	13:	IF bAutoModeOn AND  bISealingSeparatorXAxisHome AND  bISealingTopPistonHome AND bISealingBottomPistonHome AND bISealingSeparatorYAxisHome  THEN
		bSaelUnitIntOver:=TRUE;
		step:=step+1;
		END_IF

	14:	bSealingUnitIntOver:=TRUE;
		step:=step+1;



	15:	step:=0;



END_CASE

IF bFwdRevPistonRst THEN bQRForwardPistonValve:=TRUE; bQRReversePistonValve:=TRUE; END_IF

IF bIForwardPistonEnd AND bIReversePistonEnd THEN bFwdRevPistonRst:=FALSE; bQRForwardPistonValve:=FALSE; bQRReversePistonValve:=FALSE; END_IF

IF NOT bIEmergencySwitch OR bStopHmi  OR bServoOff  OR bIMcStop THEN

		bQMWrappingChannelPistonValve1:=FALSE;
		bQMWrappingChannelPistonValve2:=FALSE;
		bQMWrappingChannelPistonValve3:=FALSE;
		bQMForwardPistonValve:=FALSE;
		bQMReversePistonValve:=FALSE;
		bAWrappingCone123OnAuto:=FALSE;
		bAWrappingCone123_23OnAuto:=FALSE;
		bAWrappingCone3OnAuto:=FALSE;
		bAWrappingCone23OnAuto:=FALSE;
		bAWrappingCone23OnAuto1:=FALSE;
		bQAForwardPistonValve:=FALSE;
		bQAReversePistonValve:=FALSE;
		bAInitializeSeq:=FALSE;
		bFwdRevPistonRst:=FALSE;
		bARWrappingCone123OnRst:=FALSE;
		bARWrappingCone123FwdCom:=FALSE;
		bAR3ConeWrappOver:=FALSE;
		tA3ConesealStartDly(IN:=FALSE);
		bQRSealingSeparatorXAxisPistonValve:=FALSE;
		bQRSealingSeparatorYAxisPistonValve:=FALSE;
		bQRSealingTopPistonValve:=FALSE;
		bQRSealingTopPistonValve:=FALSE;
		bSaelUnitIntOver:=FALSE;
		step:=0;

END_IF
END_PROGRAM

(* POU Auto/Sealing_Conveyor_23, ST *)
PROGRAM Sealing_Conveyor_23
VAR

	bA3ConeSealStarted23: BOOL;
	bQASealingConveyor1_23: BOOL;
	bQASealingConveyor2_23: BOOL;
	ConvStopDly1_23: TON;
	bA3ConeSealComp23: BOOL;
	step1: INT;
	CTU_1_23: CTU;
	bAConeCountSenEnable1_23: BOOL;
	bA6thConeSealStarted23: BOOL;
	bA6thConeSealComp23: BOOL;
	ConvStopDly2_23: TON;
	step2: INT;
	step3: INT;
	bSealConvIntOverTemp: BOOL;
	bStopHmitemp: BOOL;
	ConeMissChk_1: RS_Error;
	ConeMissErr_1: BOOL;
	ConeMissChk_2: RS_Error;
	ConeMissErr_2: BOOL;
	ConeMissbit: BOOL;
	SealingStep: INT;
	Timer1: TON;
	Timer2: TON;
	Timer3: TON;
	Timer4: TON;
	bAPauseEnable: BOOL;

	bConeMissBit1: BOOL;
	bConeMissBit2: BOOL;
	bConeMissBit3: BOOL;
	bQASealingConveyor3_23: BOOL;
	tSealStopDly: TIME;
	SealingStep2: INT;
	Timer5: TON;
	Timer6: TON;
	Timer7: TON;
	bConeMissBit11: BOOL;
	bConeMissBit22: BOOL;
	bConeMissBit33: BOOL;
	bConeMissBitSec: BOOL;
	tSealStopDlySec: TIME;
	ConeMissMonitorbit: BOOL;
	bAConeMissAtSealConv: BOOL;
	bAConeMissAtSealConv2: BOOL;
	SingleStep: INT;
	TON_6: TON;
	bAConeCountSenSensed: BOOL;
	bAConeCountSenSensedOff: BOOL;
	R_TRIG_3: R_TRIG;
	R_TRIG_9: R_TRIG;
	CTU_AlarmOnly: CTU;
	bCountLock1: BOOL;
	bCountLock2: BOOL;
	bCountLock: BOOL;
	bAConeMissAtSealConv3: BOOL;
	bQASealingConveyor4_23: BOOL;
	bQASealingConveyor5_23: BOOL;
	bAConeMissAtSealConv4: BOOL;
	bQASealingConveyor6_23: BOOL;
	bCountLock3: BOOL;
	bCountLock4: BOOL;
	bCountLock5: BOOL;
	bCountLock6: BOOL;
	bCountLockBit: BOOL;
	bSet1Started: BOOL;
	bSecSetStarted: BOOL;
	SealCountBit2: BOOL;
END_VAR
bQASealingConveyorMotor2:= ((bQASealingConveyor1_23 OR bQASealingConveyor2_23 OR  bQASealingConveyor3_23 OR bQASealingConveyor5_23 OR bQASealingConveyor4_23 OR bQASealingConveyor6_23 )) ;


CASE step1 OF

	0:	IF bAutoModeOn AND b2_3SetHmiSelected AND   bA3ConeWrappOver AND bQASealingSeparatorYAxisPistonValve THEN
		CTU_1_23.RESET:=TRUE;
		CTU_AlarmOnly.RESET:=TRUE;
		bA3ConeSealStarted23:=TRUE;
		ConvStopDly1_23(IN:=FALSE);
		tSealStopDly:=t#2.5s;
		step1:=step1+1;
		END_IF

	1:	IF NOT bAPauseSeq THEN step1:=step1+1; END_IF


	2:	IF bAutoModeOn AND b2_3SetHmiSelected AND  bA3ConeSealStarted23 AND bISealingSeparatorXAxisEnd THEN
		bA3ConeSealComp23:=TRUE;
		CTU_1_23.RESET:=FALSE;
		CTU_AlarmOnly.RESET:=FALSE;
		 Timer1(IN:=FALSE);
		step1:=step1+1;
		END_IF

	3:	step1:=step1+1;

	4:	IF bAutoModeOn AND   bA3ConeSealComp23  AND (bSealConvStart1 OR bSealConvStart3 ) AND  NOT bAPauseSeq  AND NOT bASealSepaX_axisRsError THEN
		bQASealingConveyor1_23:=TRUE;
		bSet1Started:=TRUE;
		step1:=step1+1;
		END_IF

	5:	ConvStopDly1_23(IN:=FALSE); step1:=step1+1;


	6:	IF CTU_1_23.CV>=3 THEN
		bSealConvStart1:=FALSE;
		bSealConvStart3:=FALSE;
		bA3ConeSealComp23:=FALSE;
		bA3ConeSealStarted23:=FALSE;
		bA3COneCrossed:=TRUE;
		step1:=step1+1;
		END_IF

	7:	step1:=step1+1;

	8:	IF bIColumnconeDetection THEN
		step1:=step1+1;
		END_IF

	9:	step1:=step1+1;


	10:	ConvStopDly1_23(IN:=TRUE , PT:= tSealStopDly , Q=> , ET=> );
		IF ConvStopDly1_23.Q THEN    step1:=step1+1; END_IF


	11:	 step1:=step1+1;

	12:	bQASealingConveyor1_23:=FALSE;
		bA3COneCrossed:=FALSE;
		bQASealingConveyor3_23:=FALSE;
		bQASealingConveyor5_23:=FALSE;
		bQASealingConveyor6_23:=FALSE;
		bAColumnPushPistonStart1_23:=TRUE;
		bASealConvEnd1:=TRUE;
		bCountLock1:=FALSE;
		bCountLock5:=FALSE;
		bCountLock6:=FALSE;
		bSet1Started:=FALSE;
		bCountLockBit:=FALSE;
		step1:=step1+1;

	13:	 step1:=step1+1;


	14:	step1:=0;

END_CASE

IF bQASealingConveyorMotor AND bSet1Started  AND CTU_1_23.CV=3 THEN bCountLockBit:=TRUE; END_IF


IF bQASealingConveyorMotor AND bIConeCountSensor AND b2_3SetHmiSelected AND NOT bCountLockBit AND NOT SealCountBit2  THEN
bAConeCountSenEnable1_23:=TRUE;
ELSE
bAConeCountSenEnable1_23:=FALSE;
END_IF

CTU_1_23(
	CU:=bAConeCountSenEnable1_23 ,
	RESET:= ,
	PV:=6 ,
	Q=> ,
	CV=> );

CTU_AlarmOnly(
	CU:=(bAConeCountSenEnable1_23 AND NOT bCountLock) ,
	RESET:= ,
	PV:=6 ,
	Q=> ,
	CV=> );




CASE step2 OF

	0:	IF bAutoModeOn AND b2_3SetHmiSelected AND  bA6ConeWrappOver23 AND bQASealingSeparatorYAxisPistonValve  THEN
		bA6thConeSealStarted23:=TRUE;
		ConvStopDly2_23(IN:=FALSE);
		tSealStopDlySec:=t#2.5s;
		step2:=step2+1;
		END_IF

	1:	step2:=step2+1;


	2:	 IF   bISealingSeparatorXAxisEnd THEN
		step2:=step2+1;
		END_IF

	3:	 step2:=step2+1;


	4:	IF bAutoModeOn AND b2_3SetHmiSelected  AND bAFirstSetToMatrix   THEN
		bA6thConeSealComp23:=TRUE;
		Timer2(IN:=FALSE); 															(*===============	bAFirstSetToMatrix:=FALSE; ============= Removed for interlock  Checking========= *)
		step2:=step2+1;
		END_IF


	5:	step2:=step2+1;

	6:	IF bAutoModeOn AND   bA6thConeSealComp23  AND  bSealConvStart2 AND  NOT bAPauseSeq THEN
		bQASealingConveyor2_23:=TRUE;
		bSecSetStarted:=TRUE;
		step2:=step2+1;
		END_IF

	7:	ConvStopDly2_23(IN:=FALSE); step2:=step2+1;

	8:	IF CTU_1_23.CV>=6 THEN
		bSealConvStart2:=FALSE;
		bA6thConeSealComp23:=FALSE;
		bA6thConeSealStarted23:=FALSE;
		bA6ConeCrossed:=TRUE;
		step2:=step2+1;
		END_IF

	9:	 step2:=step2+1;

	10:	IF bIColumnconeDetection THEN
		step2:=step2+1;
		END_IF

	11:	 step2:=step2+1;

	12:	ConvStopDly2_23(IN:=TRUE , PT:=tSealStopDlySec , Q=> , ET=> );
		IF ConvStopDly2_23.Q THEN   step2:=step2+1; END_IF

	13:	 step2:=step2+1;

	14:	 CTU_1_23.RESET:=TRUE;
		   step2:=step2+1;

	15:	 step2:=step2+1;

	16:	bQASealingConveyor2_23:=FALSE;
		bQASealingConveyor3_23:=FALSE;
		bQASealingConveyor4_23:=FALSE;
		bA6ConeCrossed:=FALSE;
		bAColumnPushPistonStart2_23:=TRUE;
		bASealConvEnd2:=TRUE;
		bCountLock2:=FALSE;
		bCountLock3:=FALSE;
		bCountLock4:=FALSE;
		SealCountBit2:=FALSE;
		bSecSetStarted:=FALSE;
		  step2:=step2+1;

	17:	 step2:=step2+1;

	18:	CTU_1_23.RESET:=FALSE;
		step2:=0;


END_CASE


IF bQASealingConveyorMotor AND bSecSetStarted AND  CTU_1_23.CV=6 THEN SealCountBit2:=TRUE; END_IF


(*================ Sealing Conveyor Start Condition=============*)


IF bRowStopperIntOver THEN
bSealConvIntOverTemp:=TRUE;
END_IF




CASE step3 OF


0:	IF bSealConvIntOverTemp  AND b2_3SetHmiSelected  THEN
	Step3:=Step3+1;
	END_IF

1:	IF NOT bIColumnconeDetection THEN
	bSealConvStart1:=TRUE;
	Step3:=Step3+1;
	END_IF

2:	IF  CTU_1_23.CV=3 THEN

	Step3:=Step3+1;
	END_IF

3:	IF bIColumnconeDetection THEN
	Step3:=Step3+1;
	END_IF

4:	IF bAFirstSetToMatrix  THEN
	bSealConvStart2:=TRUE;
	Step3:=Step3+1;
	END_IF

5:	IF	CTU_1_23.CV=6 THEN
	bAFirstSetToMatrix:=FALSE;
	Step3:=Step3+1;
	END_IF

6:	IF bIColumnconeDetection THEN
	Step3:=Step3+1;
	END_IF

7:	IF bASecondSetToMatrix THEN
	bSealConvStart3:=TRUE;
	Step3:=Step3+1;
	END_IF

8:	bASecondSetToMatrix:=FALSE;
	Step3:=1;
END_CASE

(*

	IF bSealConvStart1 OR bSealConvStart2 OR bSealConvStart2 THEN
	bAConvReady:=TRUE;
	ELSE
	bAConvReady:=FALSE;
	END_IF
*)
(*=================================Stop Logic=====================*)



IF bQASealingConveyor1_23 AND CTU_AlarmOnly.CV =3  THEN  bCountLock1:=TRUE; END_IF

IF bQASealingConveyor5_23 AND CTU_AlarmOnly.CV =3  THEN  bCountLock5:=TRUE; END_IF

IF bQASealingConveyor6_23 AND CTU_AlarmOnly.CV =3  THEN  bCountLock6:=TRUE; END_IF


IF bQASealingConveyor2_23 AND CTU_AlarmOnly.CV =6  THEN  bCountLock2:=TRUE; END_IF


IF bQASealingConveyor3_23 AND CTU_AlarmOnly.CV =6  THEN  bCountLock3:=TRUE; END_IF


IF bQASealingConveyor4_23 AND CTU_AlarmOnly.CV =6  THEN  bCountLock4:=TRUE; END_IF


 IF bCountLock1 OR bCountLock2 OR  bCountLock3 OR bCountLock4 OR  bCountLock5 OR bCountLock6 THEN bCountLock:=TRUE; ELSE bCountLock:=FALSE; END_IF



IF bQASealingConveyor1_23  AND  bIColumnconeDetection  AND  (CTU_AlarmOnly.CV ) <3  THEN
bAConeMissAtSealConv:=TRUE; SealConeMiss:=' Cone  Missing From Sealing Conveyor';  bQASealingConveyor1_23:=FALSE;  END_IF
(*IF  THEN bAConeMissAtSealConv:=TRUE;  SealConeMiss:=' Cone  Missing From Sealing Conveyor'; bQASealingConveyor1_23:=FALSE; tSealStopDly:=t#4s;
ELSE   SealConeMiss:='Continue Machine Operation'; END_IF *)
IF bAConeMissAtSealConv AND bErrorReset THEN
 bQASealingConveyor5_23:=TRUE;  Step1:=5;  tSealStopDly:=t#4s;    SealConeMiss:='Continue Machine Operation'; bAConeMissAtSealConv:=FALSE; END_IF



IF bQASealingConveyor5_23  AND  bIColumnconeDetection  AND  (CTU_AlarmOnly.CV ) <3  THEN
bAConeMissAtSealConv4:=TRUE; SealConeMiss:=' Cone  Missing From Sealing Conveyor';  bQASealingConveyor5_23:=FALSE;  END_IF
(*IF bQASealingConveyor3_23 AND (CTU_1_23.CV )=3 THEN bAConeMissAtSealConv:=FALSE;  END_IF*)
IF bAConeMissAtSealConv4 AND bErrorReset THEN
bQASealingConveyor6_23:=TRUE;  Step1:=5;  tSealStopDly:=t#4s;    SealConeMiss:='Continue Machine Operation'; bAConeMissAtSealConv4:=FALSE; END_IF




IF bQASealingConveyor2_23 AND  bIColumnconeDetection AND   (CTU_AlarmOnly.CV ) >=3 AND   (CTU_AlarmOnly.CV ) <6 THEN
bAConeMissAtSealConv2:=TRUE; SealConeMiss:=' Cone  Missing From Sealing Conveyor';  bQASealingConveyor2_23:=FALSE;END_IF
(*IF Timer2.Q AND  (CTU_AlarmOnly.CV ) <=6 AND  (CTU_1_23.CV ) >=3 THEN bAConeMissAtSealConv2:=TRUE;  SealConeMiss:=' Cone  Missing From Sealing Conveyor'; bQASealingConveyor2_23:=FALSE; tSealStopDlySec:=t#4s; ELSE   SealConeMiss:='';END_IF*)
IF bAConeMissAtSealConv2 AND bErrorReset THEN
 bQASealingConveyor3_23:=TRUE; Step2:=7; tSealStopDlySec:=t#4s;   SealConeMiss:='Continue Machine Operation'; bAConeMissAtSealConv2:=FALSE; END_IF

(*IF bQASealingConveyor3_23 AND (CTU_1_23.CV )=6 THEN bAConeMissAtSealConv2:=FALSE;  END_IF *)


IF bQASealingConveyor3_23 AND  bIColumnconeDetection AND   (CTU_AlarmOnly.CV ) >=3 AND   (CTU_AlarmOnly.CV ) <6 THEN
  bAConeMissAtSealConv3:=TRUE; SealConeMiss:=' Cone  Missing From Sealing Conveyor';  bQASealingConveyor3_23:=FALSE;END_IF
IF bAConeMissAtSealConv3 AND bErrorReset THEN
 bQASealingConveyor4_23:=TRUE; Step2:=7; tSealStopDlySec:=t#4s;   SealConeMiss:='Continue Machine Operation'; bAConeMissAtSealConv3:=FALSE; END_IF


IF bAConeMissAtSealConv OR bAConeMissAtSealConv3 OR bAConeMissAtSealConv2 OR bAConeMissAtSealConv4  THEN
SealBitAlert:=TRUE; ELSE SealBitAlert:=FALSE; END_IF


IF NOT bIEmergencySwitch OR bStopHmi   OR bServoOff  OR bIMcStop   THEN
CTU_1_23.RESET:=TRUE;
CTU_AlarmOnly.RESET:=TRUE;
ConvStopDly1_23(IN:=FALSE);
bA3ConeSealComp23:=FALSE;
bQASealingConveyor1_23:=FALSE;
bA3COneCrossed:=FALSE;
bAColumnPushPistonStart1_23:=FALSE;
bASealConvEnd1:=FALSE;
bCountLock1:=FALSE;
bCountLock5:=FALSE;
bCountLock6:=FALSE;
bAConeCountSenEnable1_23:=FALSE;
bA6thConeSealStarted23:=FALSE;
ConvStopDly2_23(IN:=FALSE);
bA6thConeSealComp23:=FALSE;
Timer2(IN:=FALSE);
bAColumnPushPistonStart2_23:=FALSE;
bASealConvEnd2:=FALSE;
bCountLock2:=FALSE;
bCountLock3:=FALSE;
bCountLock4:=FALSE;
bSealConvIntOverTemp:=FALSE;
bSealConvStart1:=FALSE;
bSealConvStart2:=FALSE;
bAFirstSetToMatrix:=FALSE;
bSealConvStart3:=FALSE;
bASecondSetToMatrix:=FALSE;
bCountLock:=FALSE;
bAConeMissAtSealConv:=FALSE;
bQASealingConveyor5_23:=FALSE;
bAConeMissAtSealConv4:=FALSE;
bQASealingConveyor6_23:=FALSE;
bQASealingConveyor4_23:=FALSE;
bAConeMissAtSealConv2:=FALSE;
bQASealingConveyor3_23:=FALSE;
SealBitAlert:=FALSE;
bAConeMissAtSealConv3:=FALSE;
step1:=0;
step2:=0;
Step3:=0;

ELSE
CTU_1_23.RESET:=FALSE;
CTU_AlarmOnly.RESET:=FALSE;

END_IF
END_PROGRAM

(* POU Auto1/ConeFeedPiston_23, ST *)
PROGRAM ConeFeedPiston_23
VAR

	R_TRIG_1: R_TRIG;
	CounterTiltRst: BOOL;
	step: INT;

	ConeFeedConvFwdDly1: TON;
	CounterTilt23Rst: BOOL;
	CounterTilt23Rst_R_TRIG: R_TRIG;

	bAConeFeedFwdStart23: BOOL;
	CTU_1: CTU;
	test: BOOL;
	CounterTilt23Enable: BOOL;

	CounterTilt23Rst_TRIG: R_TRIG;

	bIForwardPistonHometemp: BOOL;
	bIReversePistonHometemp: BOOL;
	bITiltingEndtemp: BOOL;
	bITiltingHometemp: BOOL;


	bErrorCheckBit1: BOOL;

	tFwdRSErrCheckDly: TON;
	FwdRevCylHomeChk: RS_Error;
	FwdRevCylHomeSenOk: BOOL;
	FwdRevCylHomeSenErr: BOOL;
	testtemp: BOOL;
	Timer1: TON;
	CTUtEST: CTU;
	CTUtESTcv: INT;
	bAUnitBConeCrossingOff: BOOL;
	step2: INT;
	R_TRIG_3: R_TRIG;
	TON_6: TON;
	bAUnitBConeCrossing_3: BOOL;
	bAUnitBConeCrossingOff_3: BOOL;
	R_TRIG_23: R_TRIG;
	bAfeedingConvOn: BOOL;
END_VAR
IF  NOT bIEmergencySwitch OR bServoOff OR bIMcStop OR   bStopHmi  THEN
	bAConeFeedFwdStart23:=FALSE;
	CounterTiltRst:=TRUE;
	CounterTilt23Rst1:=TRUE;
	bQAConeFeedingPistonOnAuto1:=FALSE;
	CounterTilt23Enable:=FALSE;
	bErrorCheckBit1:=FALSE;
	Timer1(IN:=FALSE);
	FwdRevCylHomeSenOk:=FALSE;
	ConeFeedConvFwdDly1(IN:=FALSE);
	TON_6(IN:= FALSE);
	bAUnitBConeCrossing_3 :=FALSE;
	bAFeedingConvOff:=FALSE;
	step:=0;
	step2:=0;
	ELSE
	CounterTilt23Rst1:=FALSE;
	CounterTiltRst:=FALSE;
END_IF



(*==================== Cone Feeding Piston Logic For 2*3 Model==================*)




IF  b2_3SetHmiSelected AND bAutoModeOn AND ConeFeedConvFwdDly1.Q  AND bIConeFeedingPistonHome   AND  NOT bQAFeedingConveyorMotor
 AND bIForwardPistonHome AND bIReversePistonHome   AND  NOT bAPauseSeq     THEN
		bQAConeFeedingPistonOnAuto1:=TRUE;
END_IF

IF   b2_3SetHmiSelected AND  bQAConeFeedingPistonValve AND bAutoModeOn AND   bIConeFeedingPistonEnd AND  NOT bAPauseSeq
 AND NOT bAConeFeddCylFwdRsError  THEN
		bQAConeFeedingPistonOnAuto1:=FALSE;
END_IF


c18_ConeCounter1(
	CU:=CounterTilt23Enable,
	RESET:=,
	PV:= 18,
	Q=> ,
	CV=> );

CounterTilt23(
	CU:=bAUnitBConeCrossing_3,
	RESET:=CounterTilt23Rst  OR CounterTilt23Rst1,
	PV:= 6,
	Q=> ,
	CV=>CounterTilt23_CV_HMI );
(*

CTUtEST(
	CU:=CounterTilt23Enable ,
	RESET:= ,
	PV:= 56,
	Q=> ,
	CV=>CTUtESTcv );

*)


R_TRIG_23(CLK:=bQAFeedingConveyorMotor , Q=> );
IF R_TRIG_23.Q THEN bAfeedingConvOn:=TRUE; END_IF

IF bIConeOrientationTop  AND b2_3SetHmiSelected AND bQAFeedingConveyorMotor AND bIConeFeedingPistonHome   THEN

CounterTilt23Enable:=TRUE;

ELSE(* IF NOT bAPauseSeq THEN *)
CounterTilt23Enable:=FALSE;
END_IF


R_TRIG_1(CLK:= bIConeOrientationTop , Q=> );


ConeFeedConvFwdDly1(IN:=bAConeFeedFwdStart23 , PT:=t#1s , Q=> , ET=> );  (* ===old Value  PT:=t#1s *)




CASE step OF

	0:	IF CounterTilt23.CV=1AND bIForwardPistonHome AND bIReversePistonHome AND NOT bITiltingEnd  AND bITiltingHome
		AND NOT bAResetEnabled AND bATiltPistonInHome THEN
		bAConeFeedFwdStart23:=TRUE;
		bErrorCheckBit1:=TRUE;
		step:=step+1;
		END_IF sMessage_23_Feeding:='Check Forward , Reverse & Tilting Piston Home Reed Switch ';

	1:	 step:=step+1;

	2:	IF bAutoModeOn AND  bIConeFeedingPistonEnd  AND  NOT bFeedinfCylFwdRsError THEN
		bAConeFeedFwdStart23:=FALSE;
		bATiltPistonInHome:=FALSE;
		bErrorCheckBit1:=FALSE;
		step:=step+1;
		END_IF

	3:	 step:=step+1;

	4:	IF   CounterTilt23.CV = 2  AND bIForwardPistonHome AND bIReversePistonHome  AND bAConeFeedCylStart   AND bITiltingHome AND  NOT bAPauseSeq  THEN
		 bAConeFeedFwdStart23:=TRUE ;
		bErrorCheckBit1:=TRUE;
		IF NOT bIConeFeedingPistonHome THEN
		step:=step+1;
		END_IF
		END_IF sMessage_23_Feeding:='Check Forward , Reverse & Tilting Piston Home Reed Switch ';

	5:	 step:=step+1;

	6:  IF  bAutoModeOn AND bIConeFeedingPistonEnd AND  NOT bFeedinfCylFwdRsError THEN
		bErrorCheckBit1:=FALSE;
		bAConeFeedFwdStart23:=FALSE;
		bAConeFeedCylStart:=FALSE;
		step:=step+1;
		END_IF

	7:	 step:=step+1;


	8:     IF  CounterTilt23.CV = 3 AND bIForwardPistonHome AND bIReversePistonHome AND bITiltingEnd  AND  NOT bAPauseSeq    THEN
		bAConeFeedFwdStart23:=TRUE;
		bErrorCheckBit1:=TRUE;
		step:=step+1;
		END_IF sMessage_23_Feeding:='Check Forward  & Reverse  Piston Home Reed Switch ';

	9:	 step:=step+1;

	10:	IF bAutoModeOn AND  bIConeFeedingPistonEnd AND  NOT bFeedinfCylFwdRsError THEN
		bAConeFeedFwdStart23:=FALSE;
		bErrorCheckBit1:=FALSE;
		step:=step+1;
		END_IF


	11:	step:=step+1;

	12:	IF CounterTilt23.CV = 4 AND bIForwardPistonHome AND bIReversePistonHome    AND bA4thConeFeedStartAuto23
		 AND bITiltingHome  AND  NOT bAPauseSeq   THEN
		bAConeFeedFwdStart23:=TRUE;
		bErrorCheckBit1:=TRUE;
		step:=step+1;
		END_IF sMessage_23_Feeding:='Check Forward ,Reverse & Tilting Piston Home Reed Switch ';

	13:	 step:=step+1;

	14:	IF bAutoModeOn AND  bIConeFeedingPistonEnd AND  NOT bFeedinfCylFwdRsError THEN
		bAConeFeedFwdStart23:=FALSE;
		bErrorCheckBit1:=FALSE;
		bA4thConeFeedStartAuto23:=FALSE;
		step:=step+1;
		END_IF

	15:	step:=step+1;

	16:	IF   CounterTilt23.CV = 5  AND bIForwardPistonHome AND bIReversePistonHome  AND bITiltingEnd    AND  NOT bAPauseSeq    THEN
		bAConeFeedFwdStart23:=TRUE;
		bErrorCheckBit1:=TRUE;
		step:=step+1;
		END_IF sMessage_23:='Check Forward & Reverse Piston Home Reed Switch ';

	17:	 step:=step+1;

	18:	IF bIConeFeedingPistonEnd  AND  NOT bFeedinfCylFwdRsError THEN
		bAConeFeedFwdStart23:=FALSE;
		bErrorCheckBit1:=FALSE;
		step:=step+1;
		END_IF


	19:	Timer1(IN:=FALSE);
		 step:=step+1;



	20: IF   CounterTilt23.CV = 6  AND bIForwardPistonHome AND bIReversePistonHome AND bA6thConeFeedStartAuto23   AND  NOT bAPauseSeq    THEN
		Timer1(IN:=TRUE , PT:=t#0.5s , Q=> , ET=> );
		bErrorCheckBit1:=TRUE;
		IF  Timer1.Q THEN bA6thConeFeedStart23:=FALSE;  step:=step+1; END_IF
		END_IF sMessage_23:='Check Forward  & Reverse   Piston Home Reed Switch ';


	21:	bAConeFeedFwdStart23:=TRUE;
		 step:=step+1;

	22:	IF bIConeFeedingPistonEnd AND  NOT bFeedinfCylFwdRsError THEN
		bAConeFeedFwdStart23:=FALSE;
		Timer1(IN:=FALSE);
		bErrorCheckBit1:=FALSE;
		 step:=step+1;
		END_IF

	23:	step:=step+1;

	24:	CounterTilt23Rst:=TRUE;
		bA6thConeFeedStartAuto23:=FALSE;
		step:=step+1;

	25:	step:=step+1;

	26:	CounterTilt23Rst:=FALSE;
		step:=0;

END_CASE

(*===========Cone crossing sensor single sensing logic for UnitA side======================*)


CASE step2 OF

	0:	R_TRIG_3(CLK:=CounterTilt23Enable , Q=> );
		IF R_TRIG_3.Q THEN TON_6(IN:= FALSE); step2:=step2+1; END_IF


	1:	bAFeedingConvOff:=TRUE; TON_6(IN:= FALSE);
		step2:=step2+1;


	2:	IF NOT bAPauseSeq THEN   bAUnitBConeCrossing_3 :=TRUE;
		 step2:=Step2+1;END_IF

	3:	 step2:=step2+1;

	4: 	TON_6(IN :=  TRUE  , PT:=t#1.3s , Q=> , ET=> );
		IF TON_6.Q THEN  step2:=step2+1; END_IF


	5:	 step2:=step2+1;

	6:	bAUnitBConeCrossingOff_3:=TRUE;
		TON_6(IN:= FALSE);
		step2:=step2+1;

	7:	 step2:=step2+1;

	8:	IF bAUnitBConeCrossingOff_3 THEN bAUnitBConeCrossing_3:=FALSE; step2:=step2+1; END_IF

	9:	IF NOT bAPauseSeq THEN bAUnitBConeCrossingOff_3:=FALSE;
		 step2:=step2+1; END_IF


	10:  IF bIConeFeedingPistonEnd THEN
		step2:=Step2+1; END_IF

	11:	 IF bIConeFeedingPistonHome THEN bAFeedingConvOff:=FALSE; step2:=0; END_IF sMessage_23_Feeding:='Check Cone Feeding Piston Home Reed Switch ';

END_CASE
END_PROGRAM

(* POU Auto1/Tilt_Piston_23, ST *)
PROGRAM Tilt_Piston_23
VAR
	CounterTiltRst: BOOL;
	step: INT;
	bATiltPistonFwdStart23: BOOL;
	test1: BOOL;
	bAConeFeedingStarted23: BOOL;
	bAfeedingCom23: BOOL;
	bAFeedingRev23: BOOL;
	NotbAFeedingRev23: BOOL;
	TiltCylFwdRsErrChk: RS_Error;
	TiltCylFwdRsErr: BOOL;
	bAtiltGoHome2_23temp: BOOL;
END_VAR
	(*===========Cone Tilting Piston Reset Logic===========*)


		IF bRTiltPistonReset  AND bIForwardPistonHome AND bIReversePistonHome THEN
		step:=0;
		CounterTilt23.RESET:=TRUE;
		bATiltPistonFwdStart23:=FALSE;
		bAConeFeedingStarted23:=FALSE;
		bAfeedingCom23:=FALSE;
		bAFeedingRev23:=FALSE;
		NotbAFeedingRev23:=FALSE;
		bA4thConeFeedStartAuto23:=FALSE;
		bA4thConeFeedStart23:=FALSE;;
		bA6thConeFeedStartAuto23:=FALSE;
		bATiltPistonInHome:=FALSE;

		ELSE
		CounterTilt23.RESET:=FALSE;
		END_IF

CASE step OF

	0:	IF  CounterTilt23.CV=1 AND NOT bIConeFeedingPistonEnd AND bIConeFeedingPistonHome   AND bAutoModeOn   AND bIForwardPistonHome AND bIReversePistonHome AND NOT bAPauseSeq   THEN
		bATiltPistonFwdStart23:=FALSE;
		step:=step+1;
		END_IF  sMessage_23_Tilting:='Check Forward and Reverse Piston Home Reed Switch';

	1:	IF bITiltingHome AND NOT bITiltingEnd THEN bATiltPistonInHome:=TRUE; step:=step+1; END_IF

	2: IF  CounterTilt23.CV=2 AND   bAFeedingRev23   AND bIForwardPistonHome AND bIReversePistonHome AND NOT bAPauseSeq
		 AND NOT bAConeFeddCylFwdRsError   THEN
		bATiltPistonFwdStart23:=TRUE;
		step:=step+1;
		END_IF sMessage_23_Tilting:='Check Forward and Reverse Piston Home Reed Switch';

	3:	 step:=step+1;

	4:	 IF  CounterTilt23.CV=3  AND bIForwardPistonHome AND bIReversePistonHome AND NOT bAPauseSeq   THEN
		bATiltPistonFwdStart23:=TRUE;
		step:=step+1;
		END_IF sMessage_23_Tilting:='Check Forward and Reverse Piston Home Reed Switch';

	5:	 step:=step+1;

	6:  IF (* bAtiltGoHome1_23*)  CounterTilt23.CV= 4  AND   bIConeFeedingPistonHome AND bIForwardPistonHome AND bIReversePistonHome
		 AND bATiltEnable1 AND NOT bAPauseSeq    THEN
		bATiltPistonFwdStart23:=FALSE;
		bA4thConeFeedStart23:=TRUE;
		step:=step+1;
		END_IF sMessage_23_Tilting:='Check Forward ,  Reverse & Cone Feeding Piston Home Reed Switch';

	7:	step:=step+1;


	8:  IF  CounterTilt23.CV= 4 AND  bAFeedingRev23 AND bIForwardPistonHome AND bIReversePistonHome AND NOT bAPauseSeq   THEN
		bATiltPistonFwdStart23:=TRUE;
		step:=step+1;
		END_IF  sMessage_23_Tilting:='Check Forward and Reverse Piston Home Reed Switch';

	9:	step:=step+1;


	10:	 bATiltEnable1:=FALSE;
		step:=step+1;


	11:	step:=step+1;

	12:	IF  CounterTilt23.CV=5 AND bIConeFeedingPistonHome AND bIForwardPistonHome AND bIReversePistonHome  AND NOT bAPauseSeq  THEN
		step:=step+1;
		END_IF sMessage_23_Tilting:='Check Forward ,  Reverse & Cone Feeding Piston Home Reed Switch';


	13:	 IF NOT bConeMiss2AtWrapConv THEN  step:=step+1; END_IF

	14:	IF(* bAtiltGoHome2_23 *) CounterTilt23.CV= 6 AND bAtiltGoHome2_23 AND bIForwardPistonHome AND bIReversePistonHome
		 AND bIConeFeedingPistonHome AND NOT bAPauseSeq  AND NOT   bConeMiss2AtWrapConv THEN
		bATiltPistonFwdStart23:=FALSE;
		bA6thConeFeedStart23:=TRUE;
		step:=step+1;
		END_IF  sMessage_23_Tilting:='Check Forward ,  Reverse & Cone Feeding Piston Home Reed Switch';

	15:	 bAtiltGoHome2_23:=FALSE; step:=step+1;



	16:	IF (*CounterTilt23.CV= 6*) b2_3SetHmiSelected  AND bIConeFeedingPistonHome AND bAFeedingRev23  AND bIForwardPistonHome
		 AND bIReversePistonHome AND NOT bAPauseSeq  THEN
		bATiltPistonFwdStart23:=TRUE;
		step:=step+1;
		END_IF  sMessage_23_Tilting:='Check Forward ,  Reverse & Cone Feeding Piston Home Reed Switch';

	17:	 step:=step+1;

	18:	IF bAtiltGoHome3_23 AND bIConeFeedingPistonHome    AND bIForwardPistonHome AND bIReversePistonHome AND NOT bAPauseSeq    THEN
		bATiltPistonFwdStart23:=FALSE;
		step:=0;
		END_IF  sMessage_23_Tilting:='Check Forward ,  Reverse & Cone Feeding Piston Home Reed Switch';


END_CASE


bQAConeTiltingPistonValve2:=bATiltPistonFwdStart23;


IF bQAConeFeedingPistonValve  AND NOT NotbAFeedingRev23 THEN bAConeFeedingStarted23:=TRUE; END_IF

IF bAConeFeedingStarted23 AND bIConeFeedingPistonEnd  AND NOT NotbAFeedingRev23 THEN bAfeedingCom23:=TRUE;  END_IF

IF bAfeedingCom23 AND NOT bIConeFeedingPistonEnd AND NOT NotbAFeedingRev23 THEN bAFeedingRev23:=TRUE;  bAConeFeedingStarted23:=FALSE;   bAfeedingCom23:=FALSE;  END_IF

IF  CounterTilt23.CV= 1 OR  CounterTilt23.CV= 3 OR  CounterTilt23.CV= 5  THEN
NotbAFeedingRev23:=TRUE;
ELSE
NotbAFeedingRev23:=FALSE;
END_IF

IF bATiltPistonFwdStart23  AND bITiltingEnd THEN     bAFeedingRev23:=FALSE; END_IF



IF bA4thConeFeedStart23 AND bITiltingHome THEN
bA4thConeFeedStartAuto23:=TRUE;
END_IF


IF bA6thConeFeedStart23 AND bITiltingHome THEN
bA6thConeFeedStartAuto23:=TRUE;
END_IF
END_PROGRAM

(* POU Auto1/FwdRevPiston_2_3, ST *)
PROGRAM FwdRevPiston_2_3
VAR
	step: INT;
	bA2ndConeReached23: BOOL;
	bA3rdConeReached23: BOOL;
	bA4thConeReached23: BOOL;
	bA5thConeReached23: BOOL;
	bA6thConeReached23: BOOL;
	bA7thConeReached23: BOOL;
	bA8thConeReached23: BOOL;
	bQAForwardPistonValve23: BOOL;
	bQAReversePistonValve23: BOOL;
	test: BOOL;
	FwdCylFwdRSErrChk: RS_Error;
	FwdCylFwdRSErr: BOOL;
	RevCylFwdRSErrChk: RS_Error;
	RevCylFwdRSErr: BOOL;
	FwdCylStartBit1: BOOL;
	FwdCylSTartBit2: BOOL;
	bWrapConvReady: BOOL;
END_VAR
	(*=============================Forward and Reverse piston On/Off logic=======================*)


bQAForwardPistonValve:= ( bQAForwardPistonValve23 );

bQAReversePistonValve:= (bQAReversePistonValve23);


IF bRFwdRevPistonRst OR bAInitializeSeq    THEN
		bQAForwardPistonValve23:=FALSE;
		bQAReversePistonValve23:=FALSE;
		bA2ndConeReached23:=FALSE;
		bInterLocCounterRst:=TRUE;
		bAWrappingConvStart1_23:=FALSE;
		bA2ndConeReached23:=FALSE;
		bA3rdConeReached23:=FALSE;
		bAWrappingConvStart2_23:=FALSE;
		bAtiltGoHome1_23:=FALSE;
		bATiltEnable1:=FALSE;
		bA5thConeReached23:=FALSE;
		bA4thConeReached23:=FALSE;
		bAtiltGoHome2_23:=FALSE;
		bAWrappingConvStart3_23:=FALSE;
		bA6thConeReached23:=FALSE;
		bAtiltGoHome3_23:=FALSE;
		bAWrappingConvStart4_23:=FALSE;
		bA6conesPushedTemp:=FALSE;
		step:=0;


		ELSE
		bInterLocCounterRst:=FALSE;
END_IF




CASE step OF
	0:	IF b2_3SetHmiSelected AND NOT bQAWrappingConveyorMotor  AND NOT bCount_ConvLockBit2 AND bAutoModeOn
		 AND bWrapConvReady  (* AND CounterTilt23.CV=1 AND bITiltingHome AND bIConeFeedingPistonEnd*) AND  NOT bAPauseSeq
		 AND NOT bAConeFeddCylFwdRsError AND NOT bConeMiss4AtWrapConv   THEN
		bQAForwardPistonValve23:=TRUE;
		bInterLocCounterRst:=TRUE;
		bCone1LockBit:=FALSE;
	 (*	bA6conesPushedTemp:=FALSE;  *)
		step:=step+1;
		END_IF


	1:	 step:=step+1;

	2:	IF b2_3SetHmiSelected AND bAutoModeOn AND bIForwardPistonEnd AND  NOT bAPauseSeq AND NOT bAForwPistRsError   THEN
		bQAForwardPistonValve23:=FALSE;
		bWrapConvReady:=FALSE;
		bInterLocCounterRst:=FALSE;
		bAWrappingConvStart1_23:=TRUE;
		step:=step+1;
		END_IF

	3:	 IF  bIForwardPistonHome THEN   bAConeFeedCylStart:=TRUE;  step:=step+1; END_IF
		sMessage_23_Forwad_rev:='Check Forward Piston Home Reed Switch ';


	4:	IF CounterTilt23.CV=2 AND bIConeFeedingPistonEnd  AND  NOT bAPauseSeq  THEN
		bA2ndConeReached23:=TRUE;
	(*	bAWrappingConvStart1_23:=FALSE;  *) (*======== Changed to Wrapping unit_07.10.16=======*)
		step:=step+1;
		END_IF


	5:	 step:=step+1;

	6:	IF CounterTilt23.CV=3 AND bIConeFeedingPistonEnd  AND  NOT bAPauseSeq  THEN
		bA3rdConeReached23:=TRUE;
		step:=step+1;
		END_IF


	7:	 step:=step+1;

	8:	IF b2_3SetHmiSelected AND bAutoModeOn  AND NOT bQAWrappingConveyorMotor  AND bITiltingEnd AND bA2ndConeReached23
		AND bA3rdConeReached23  AND InterLockCounter.CV=1 AND  NOT bAPauseSeq  AND NOT bATiltPistRsError AND NOT bAConeFeddCylFwdRsError
		 AND NOT bAConeMissErrorAtWrpConv AND  NOT bACheckWrappConvError1 THEN
		bQAForwardPistonValve23:=TRUE;
		bQAReversePistonValve23:=TRUE;
		step:=step+1;
		END_IF


	9:	step:= step+1;


	10:	IF b2_3SetHmiSelected AND bAutoModeOn AND bIConeFeedingPistonHome  AND bIForwardPistonEnd AND bIReversePistonEnd
		 AND  NOT bAPauseSeq AND NOT bAForwPistRsError AND NOT bAReversPistnRsError THEN
		bQAForwardPistonValve23:=FALSE;
		bQAReversePistonValve23:=FALSE;
		bA2ndConeReached23:=FALSE;
		bA3rdConeReached23:=FALSE;
		bAWrappingConvStart2_23:=TRUE;
		(*bATiltEnable1:=TRUE;  *)
		step:=step+1;
		END_IF sMessage_23_Forwad_rev:='Check Cone Feeding Piston Home Reed Switch ';

	11:	step:=step+1;

(*-=========================mod Done here & verify============ over==========*)

	12:	 IF b2_3SetHmiSelected AND bAutoModeOn AND bIForwardPistonHome AND bIReversePistonHome  AND  NOT bAPauseSeq   THEN
		bAtiltGoHome1_23:=TRUE;
		bATiltEnable1:=TRUE;
		bAWrappingConvStart2_23:=FALSE;
		step:=step+1;
		END_IF sMessage_23_Forwad_rev:='Check Forward & Reverse Piston Home Reed Switch ';

	13:	step:=step+1;


	14:	IF b2_3SetHmiSelected AND     CounterTilt23.CV=4 AND bIConeFeedingPistonEnd  THEN
		bA4thConeReached23:=TRUE;
		step:=step+1;
		END_IF

	15:	step:=step+1;

	16:	IF b2_3SetHmiSelected AND bAutoModeOn AND NOT bQAWrappingConveyorMotor   AND  bA4thConeReached23
		 AND bITiltingEnd AND bIReversePistonHome THEN
		step:=step+1;
		END_IF sMessage_23_Forwad_rev:='Check Reverse Piston Home Reed Switch ';

	17:	step:=step+1;

	18:	IF  CounterTilt23.CV=5 AND bIConeFeedingPistonEnd THEN
		bA5thConeReached23:=TRUE;
		bAtiltGoHome1_23:=FALSE;
		step:=step+1;
		END_IF

	19:	step:=step+1;

	20:	IF b2_3SetHmiSelected AND bAutoModeOn AND NOT bQAWrappingConveyorMotor  AND( InterLockCounter.CV=3 OR bAByPassOn)
		  AND  bA5thConeReached23 AND bA4thConeReached23  AND bITiltingEnd AND bIReversePistonHome  AND bIForwardPistonHome
		 AND NOT  bATiltPistRsError AND  NOT bAPauseSeq AND NOT bAConeFeddCylFwdRsError  AND NOT bConeMiss2AtWrapConv THEN
		bQAForwardPistonValve23:=TRUE;
		bQAReversePistonValve23:=TRUE;
		step:=step+1;
		END_IF sMessage_23_Forwad_rev:='Check Forward & Reverse Piston Home Reed Switch ';

	21:	step:=step+1;

	22:	IF b2_3SetHmiSelected AND bAutoModeOn AND bIConeFeedingPistonHome  AND bIForwardPistonEnd AND bIReversePistonEnd
		AND  NOT bAPauseSeq AND NOT bAForwPistRsError AND NOT bAReversPistnRsError THEN
		bQAForwardPistonValve23:=FALSE;
		bQAReversePistonValve23:=FALSE;
		bA5thConeReached23:=FALSE;
		bA4thConeReached23:=FALSE;
		bAByPassOn:=FALSE;
		bAWrappingConvStart3_23:=TRUE;
		step:=step+1;
		END_IF sMessage_23_Forwad_rev:='Check Cone Feeding Piston Home Reed Switch ';

	23: step:=step+1;

	24:	IF bAutoModeOn AND bIForwardPistonHome  AND bIReversePistonHome AND  NOT bAPauseSeq THEN
		bAtiltGoHome2_23:=TRUE;
	(*	bAWrappingConvStart3_23:=FALSE;  *)
		step:=step+1;
		END_IF sMessage_23_Forwad_rev:='Check Forward  & Reverse Piston Home Reed Switch ';


	25:	 step:=step+1;


	26:	IF  CounterTilt23.CV=6 AND bIConeFeedingPistonEnd THEN
		bA6thConeReached23:=TRUE;
		step:=step+1;
		END_IF

	27:	step:=step+1;


	28:	IF b2_3SetHmiSelected AND bAutoModeOn AND NOT bQAWrappingConveyorMotor  AND  bA6thConeReached23   AND bITiltingEnd
		  AND bIForwardPistonHome AND( InterLockCounter.CV=5 OR bAByPassOn2 ) AND  NOT bAPauseSeq  AND NOT bATiltPistRsError
		AND NOT bAConeFeddCylFwdRsError AND NOT bConeMiss3AtWrapConv THEN
		bQAReversePistonValve23:=TRUE;
		step:=step+1;
		END_IF sMessage_23_Forwad_rev:='Check Forward Piston Home Reed Switch ';

	29:	 step:=step+1;

	30:	IF b2_3SetHmiSelected AND bAutoModeOn AND bIConeFeedingPistonHome   AND bIReversePistonEnd AND  NOT bAPauseSeq
		 AND NOT  bAReversPistnRsError THEN
		bQAReversePistonValve23:=FALSE;
		bA6thConeReached23:=FALSE;
		bAWrappingConvStart4_23:=TRUE;
		step:=step+1;
		END_IF sMessage_23_Forwad_rev:='Check Cone Feeding Piston Home Reed Switch ';

	31:	step:=step+1;


	32:	IF bAutoModeOn AND bIReversePistonHome THEN
		bAWrappingConvStart4_23:=FALSE;
		bAtiltGoHome3_23:=TRUE;
		step:=step+1;
		END_IF sMessage_23_Forwad_rev:='Check Reverse Piston Home Reed Switch ';

	33:	step:=step+1;

	34:	IF bAutoModeOn AND bITiltingHome THEN
		bAtiltGoHome3_23:=FALSE;
		step:=0;
		END_IF sMessage_23_Forwad_rev:='Check Tilting Piston Home Reed Switch ';
END_CASE

(*======================== InterLock Program for  wrong sensing of sheet or other things when second row Last cone arrived to wrapping conveyor==================*)


IF bCone1LockBit AND bA6conesPushedTemp THEN FwdCylStartBit1:=TRUE; bA6conesPushedTemp:=FALSE;
ELSIF NOT bCone1LockBit AND CounterTilt23.CV=1 AND bITiltingHome AND bIConeFeedingPistonEnd  THEN FwdCylSTartBit2:=TRUE;

END_IF
IF FwdCylStartBit1 OR FwdCylSTartBit2 THEN bWrapConvReady:=TRUE;  FwdCylStartBit1:=FALSE; FwdCylSTartBit2:=FALSE ;   END_IF
END_PROGRAM

(* POU Auto1/ConeFeedConvNew_23, ST *)
PROGRAM ConeFeedConvNew_23
VAR
	bARetUnitRunning: BOOL;
	bConePresentInConv: BOOL;
	tConeFeedConvStopDly: TON;
	step: INT;
	TON_1: TON;
	TON_2: TON;
	TON_3: TON;
	CTU_2: CTU;
	R_TRIG_2: R_TRIG;
	CTU_2Enable: BOOL;
	TON_4: TON;


	R_TRIG_1: R_TRIG;
	TON_5: TON;
	AllOutputsOn: BOOL;
	bAConveStartsAuto: BOOL;
	R_TRIG_3: R_TRIG;
	TON_6: TON;
	bAUnitBConeCrossingOff: BOOL;
	step2: INT;
	testCounter: CTU;
	testreset: BOOL;
	bConeFeedConvRst: BOOL;
	bStopHmitemp: BOOL;
	step3: INT;
	TON_7: TON;
	R_TRIG_4: R_TRIG;
	bAUnitBConeCrossingOff_2: BOOL;
	testCounter_2: CTU;
	i3ConeCountVal: INT;
	CTU_2_UB: CTU;
	i18ConeCountVal: INT;
	bConveyorStarted: BOOL;
	bConePresentInConv_1: BOOL;
END_VAR
bQAFeedingConveyorMotorA:=(bAConveStartsAuto);



IF bMCStartInAuto AND NOT  bIMcStop  AND  bIEmergencySwitch THEN
AllOutputsOn:=TRUE;
ELSE
AllOutputsOn:=FALSE;
END_IF

IF AllOutputsOn(* AND NOT bIConeOrientationTop *) AND NOT bAFeedingConvOff AND NOT bAFeedingConvOff_1  AND bIConeFeedingPistonHome AND NOT bAPauseSeq  THEN
bAConveStartsAuto:=TRUE;
ELSE
bAConveStartsAuto:=FALSE;

END_IF

(*===========Cone crossing sensor single sensing logic for UnitA side======================*)


CASE step2 OF

	0:	R_TRIG_3(CLK:=bIUnitAConeCrossing , Q=> );
		IF R_TRIG_3.Q    THEN TON_6(IN:= FALSE); step2:=step2+1; END_IF


	1:	IF  NOT bAPauseSeq THEN TON_6(IN:= FALSE);
		step2:=step2+1; END_IF


	2:	 bAUnitBConeCrossing_1 :=TRUE;
		 step2:=6;

	3:	 step2:=step2+1;

	4: 	TON_6(IN:=  TRUE  , PT:=t#1ms , Q=> , ET=> );
		IF TON_6.Q    THEN  step2:=step2+1; END_IF


	5:	 step2:=step2+1;

	6:	bAUnitBConeCrossingOff:=TRUE;
		TON_6(IN:= FALSE);
		step2:=step2+1;

	7:	 step2:=step2+1;

	8:	IF bAUnitBConeCrossingOff    THEN bAUnitBConeCrossing_1:=FALSE; step2:=step2+1; END_IF

	9:	 step2:=step2+1;

	10:	bAUnitBConeCrossingOff:=FALSE;
		step2:=0;


END_CASE







testCounter(
	CU:= bAUnitBConeCrossing_1,
	RESET:= ,
	PV:= ,
	Q=> ,
	CV=> );



 (*===============Stop Sequence===========*)


 IF NOT bIEmergencySwitch OR    bStopHmi  OR bIMcStop OR bServoOff  THEN bConeFeedConvRst:=TRUE; ELSE  bConeFeedConvRst:=FALSE;END_IF


IF bConeFeedConvRst THEN
step:=0;
bQAFeedingConveyor1_24:=FALSE;
bQAFeedingConveyor2_24:=FALSE;
bQAFeedingConveyor3_24:=FALSE;
bAConveStartsAuto:=FALSE;
bAUnitBConeCrossingOff:=FALSE;
UnitAConeCrossCount.RESET:=TRUE;
CTU_2.RESET:=TRUE;
step2:=0;
 bAUnitBConeCrossing_1 :=FALSE;
 TON_6(IN:= FALSE);
ELSE
UnitAConeCrossCount.RESET:=FALSE;
CTU_2.RESET:=FALSE;
END_IF



(*==================Logic is to Run the ConeFeed Conveyor Witout Retreival Unit===============*)

IF NOT bAAutoRetrivalEnabled AND bAutoModeOn AND bIMcStart  THEN bStartConeFeedConvInBypass:=TRUE; ELSE bStartConeFeedConvInBypass:=FALSE; END_IF
END_PROGRAM

(* POU Auto/Wrapping_Unit, ST *)
PROGRAM Wrapping_Unit
VAR

	step1: INT;

	R_TRIG_1: R_TRIG;
	Counter1: CTU;
	WrapConvStartDly: TON;
	WrapR_TRIG_1: R_TRIG;
	bAWrappingConvStartAuto2: BOOL;
	WrapR_TRIG_2: R_TRIG;
	WrapConvStartDly2: TON;

	WrapConvStartDly3: TON;
	bAWrappingConvStartAuto3: BOOL;
	WrapR_TRIG_4: R_TRIG;
	bAWrappingConvStartAuto4: BOOL;
	WrapConvStartDly4: TON;
	WrapR_TRIG_5: R_TRIG;
	bAWrappingConvStartAuto5: BOOL;
	WrapConvStartDly5: TON;
	bAWrapConeCyl1: BOOL;
	bAWrapConeCyl3: BOOL;
	bAWrapConeCyl23: BOOL;
	bASet1Comp: BOOL;
	bASet2Comp: BOOL;
	bASet: BOOL;
	bASet3Comp: BOOL;
	bA3ConeWrapStarted: BOOL;
	bA6thConeWrapStarted: BOOL;
	bA1ConeWrappOver: BOOL;
	bA2ConeWrappOver: BOOL;
	bAll3ConeWrapOver: BOOL;
	bA5ConeWrappOver: BOOL;
	bA6ConeWrappOver: BOOL;
	bA56ConeWrapOver: BOOL;
	bAWrapConeCyl23_1: BOOL;

	bATemp: BOOL;
	baConv2ndStart: BOOL;
	baConv3rdStart: BOOL;
	baConv4thStart: BOOL;
	baConv5thStart: BOOL;
	bASensorMonitorBit1: BOOL;
	bAWrappingCone123FwdCom: BOOL;
	ni: BOOL;
	step2: INT;
	bAWrappingCone3FwdCom: BOOL;
	step3: INT;
	bAWrappingCone23FwdCom: BOOL;
	step4: INT;
	bAWrappingCone23FwdCom1: BOOL;
	bASet4Comp: BOOL;
	WrapR_TRIG_3_23: R_TRIG;
	bAWrappingConvStartAuto3_23: BOOL;
	WrapConvStartDly3_23: TON;
	bAWrapConeCyl23_1_23: BOOL;
	bAWrappingCone23_23FwdCom1: BOOL;
	WrapR_TRIG_6_23: R_TRIG;
	bAWrappingConvStartAuto4_23: BOOL;
	WrapConvStartDly6_23: TON;
	bIWrappingCone: BOOL;

	bAWrappingCone123_23FwdCom: BOOL;

	step5: INT;
	bAConvRunning1: BOOL;
	bAConvRunning2: BOOL;
	TON_1: TON;
	TON_2: TON;
	bANextLayerStarted: BOOL;
	bAConvStartInterlock: BOOL;
	bAFirstConeAtWrapConv: BOOL;
	baConveyerStarted: BOOL;
	RtrigBit1: BOOL;
	R_TRIG_3: R_TRIG;
	bASensorNok: BOOL;
	WrapConvStartDlyOver: BOOL;
	test: R_TRIG;
	WrappingCone1RT: R_TRIG;
	WrappingConvRT: R_TRIG;
	WCS1Sensed: BOOL;
	TON_3: TON;
	WCS1SenseRst1: BOOL;
	TON_6: TON;
	TON_7: TON;
	TON_8: TON;
	TON_9: TON;
	TON_10: TON;
	TimerStartBit: BOOL;
	bConvRunning: BOOL;
	test1THEN: BOOL;
	test1: BOOL;
	bSaelUnitIntOverTemp: BOOL;
	step6: INT;
	step7: INT;
	bWCSStart3_24: BOOL;
	bStopHmitemp: BOOL;
	bWCSHomeSenOk: BOOL;
	WCSCylsHomeRsErrChk: RS_Error;
	WCSCylsHomeRsErr: BOOL;
	WCSCylsEndRsErrChk: RS_Error;
	bWCSHomeEndOk: BOOL;
	WCSCylsEndRsErr: BOOL;
	WCSSensorErrChk: RS_Error;
	bAWrappingConvStartAuto3_23temp: BOOL;
	bAWrappingConvStartAuto3_23temp2: BOOL;
	R_Bit1: BOOL;
	R_Bit2: BOOL;
	R_Bit3: BOOL;
	test2: BOOL;
	R_TRIG_2: R_TRIG;
	WCPReadyTemp: BOOL;
	bWrongSenChkBit: BOOL;
	WrapConvOffDly1: TON;
END_VAR
(*========================Wrapping Conveyor Logic in auto Mode=================*)

bQAWrappingConveyorMotor:= (bQAWrappingConveyorMotor1 OR bQAWrappingConveyorMotor2 OR bQAWrappingConveyorMotor3 OR bQAWrappingConveyorMotor4 OR bQAWrappingConveyorMotor5 OR bQAWrappingConveyorMotor3_23 OR bQAWrappingConveyorMotor4_23 );


(*===================Wrapping Pinston On/Off Logic In Auto Mode==================*)


bQAWrappingChannelPistonValve1:= (bAWrappingCone123OnAuto OR bAWrappingCone123_23OnAuto);

bQAWrappingChannelPistonValve2:=( bAWrappingCone123OnAuto OR bAWrappingCone23OnAuto OR bAWrappingCone23OnAuto1 OR bAWrappingCone123_23OnAuto );

bQAWrappingChannelPistonValve3:=( bAWrappingCone123OnAuto OR bAWrappingCone23OnAuto OR bAWrappingCone23OnAuto1 OR  bAWrappingCone3OnAuto OR bAWrappingCone123_23OnAuto  );


(*========================Wrapping Conveyor  Logic for First Cone in auto Mode for 2*4 and 2*3 model=================*)

WrapR_TRIG_1(CLK:= RtrigBit1 , Q=> );


IF  bAWrappingConvStart1 OR bAWrappingConvStart1_23 THEN
RtrigBit1:=TRUE;

ELSE
RtrigBit1:=FALSE;
END_IF


IF bAutoModeOn AND  WrapR_TRIG_1.Q (* OR R_TRIG_3.Q *) AND b2_3SetHmiSelected THEN  bAWrappingConvStartAuto:=TRUE; END_IF

WrapConvStartDly(IN:= bAWrappingConvStartAuto, PT:=t#1s , Q=> , ET=> );




IF bAutoModeOn AND  WrapConvStartDly.Q   AND bIWrappingChannelPiston1_Home AND bIWrappingChannelPiston2_Home
AND bIWrappingChannelPiston3_Home  AND WCPReady AND NOT bIWrappingCone1 AND NOT bIWrappingCone2 AND NOT bIWrappingCone3
AND NOT bACheckWrappConvError1 AND NOT bACheckWrappConvError4  AND b2_3SetHmiSelected  THEN
bQAWrappingConveyorMotor1:=TRUE;
bAconvReayTemp2:=FALSE;
bAconvReadyTemp5:=FALSE;
InterLockCounter.RESET:=FALSE;
bAWrappingConvStartAuto:=FALSE;
bAWrappingConvStart1_23:=FALSE;
bAConvStartBit:=TRUE;
ELSIF bAutoModeOn AND  WrapConvStartDly.Q   AND bIWrappingChannelPiston1_Home AND bIWrappingChannelPiston2_Home AND
bIWrappingChannelPiston3_Home  (*AND bWrongSenChkBit *)AND (  bIWrappingCone1 OR  bIWrappingCone2 OR  bIWrappingCone3 )
 AND NOT bACheckWrappConvError4  AND b2_3SetHmiSelected THEN
bACheckWrappConvError1:=TRUE;
ConeMissAlarm:='Check Wrapping Sensor 1_2_3';
END_IF

IF bACheckWrappConvError1 AND(  bErrorReset OR  bStopHmi ) AND b2_3SetHmiSelected AND NOT bIWrappingCone1 AND NOT  bIWrappingCone2 AND NOT  bIWrappingCone3
THEN  bACheckWrappConvError1:=FALSE; ConeMissAlarm:=''; END_IF

R_TRIG_2(CLK:=bWrpConvIntOver , Q=> );
IF R_TRIG_2.Q THEN WCPReadyTemp:=TRUE; END_IF

IF WCPReadyTemp OR bA6conesPushedTemp THEN bWrongSenChkBit:=TRUE; ELSE  bWrongSenChkBit:=FALSE; END_IF

(*
s
(*==============Wrong Cone or Sheet Sensing Error========================*)


IF  NOT  bCount_ConvLockBitTemp AND   bAutoModeOn AND  bAWrappingConvStartAuto  AND bIWrappingChannelPiston1_Home AND bIWrappingChannelPiston2_Home AND bIWrappingChannelPiston3_Home  AND WCPReady AND(  bIWrappingCone1 OR  bIWrappingCone2 OR  bIWrappingCone3 ) THEN
bACheckWrappConvError1:=TRUE;
(*ConeMissAlarm:='Check Wrapping Sensor 1 & 2 & 3'; *)
END_IF


IF bACheckWrappConvError1 AND  bErrorReset THEN  bACheckWrappConvError1:=FALSE; ConeMissAlarm:=''; END_IF

*)

(*WrapConvOffDly1(IN:= bQAWrappingConveyorMotor1, PT:=t#0.3s , Q=> , ET=> );*)

IF   bAutoModeOn AND  bIWrappingCone1 AND bAConvStartBit  AND b2_3SetHmiSelected  THEN
bQAWrappingConveyorMotor1:=FALSE; END_IF


(*===============Wrapping Conveyor 2nd and 3rd Cone  Logic  in auto Mode for 2*4 and 2*3 model==================*)

(*===============Wrapping piston 1 & 2nd and 3rd  Logic for First Cone in auto Mode  for 2*4 and 2*3 model==================*)

WrapR_TRIG_2(CLK:= ( bAWrappingConvStart2 OR bAWrappingConvStart2_23) , Q=> );


IF bAutoModeOn AND  WrapR_TRIG_2.Q THEN  (* bAWrappingConvStartAuto:=FALSE;  *) bAWrappingConvStartAuto2:=TRUE; END_IF

WrapConvStartDly2(IN:= bAWrappingConvStartAuto2, PT:=t#0.5s , Q=> , ET=> );


IF bAutoModeOn AND  WrapConvStartDly2.Q  AND bIWrappingChannelPiston1_Home AND bIWrappingChannelPiston2_Home
AND bIWrappingChannelPiston3_Home AND NOT bIWrappingCone2 AND NOT bIWrappingCone3  AND NOT bACheckWrappConvError2
AND  b2_3SetHmiSelected THEN
bQAWrappingConveyorMotor2:=TRUE;
bAWrappingConvStartAuto2:=FALSE;
bAConvRunning1:=TRUE;
ELSIF bAutoModeOn AND  WrapConvStartDly2.Q  AND bIWrappingChannelPiston1_Home AND bIWrappingChannelPiston2_Home
AND bIWrappingChannelPiston3_Home AND ( bIWrappingCone2 OR  bIWrappingCone3 ) AND b2_3SetHmiSelected  THEN
bACheckWrappConvError2:=TRUE;
ConeMissAlarm:='Check Wrapping Sensor  2_3';
END_IF

IF bACheckWrappConvError2 AND (bErrorReset  OR  bStopHmi) AND b2_3SetHmiSelected  AND NOT  bIWrappingCone2 AND NOT bIWrappingCone2   THEN bACheckWrappConvError2:=FALSE; ConeMissAlarm:='';  END_IF

IF  bAutoModeOn AND bAConvRunning1  (* AND  bIWrappingCone1 AND bIWrappingCone2   *)AND bIWrappingCone3 THEN
bQAWrappingConveyorMotor2:=FALSE;
  (*bAWrappingConvStartAuto2:=FALSE;  *)
bWrapConvStopped2:=TRUE;
 (*  bAWrapConeCyl123:=TRUE;  *)


END_IF

(*

(*===============Wrong Cone Or Sheet sensing error=====================*)
IF bAutoModeOn AND  bAWrappingConvStartAuto2  AND bIWrappingChannelPiston1_Home AND bIWrappingChannelPiston2_Home AND bIWrappingChannelPiston3_Home AND ( bIWrappingCone2 OR  bIWrappingCone3 ) THEN
bACheckWrappConvError2:=TRUE;
(*ConeMissAlarm:='Check Wrapping Sensor  2 & 3';  *)
END_IF

IF bACheckWrappConvError2 AND bErrorReset THEN bACheckWrappConvError2:=FALSE; ConeMissAlarm:='';  END_IF


*)


(*===============Wrapping piston 123 on/off logic  for 2*4 and 2*3 model =======Cones 1 2 3=============*)
CASE step1 OF

	0:	TON_1(IN:= FALSE);
		step1:=step1+1;

	1:	step1:=step1+1;

	2:	IF bAutoModeOn AND  bAWrapConeCyl123 AND b2_3SetHmiSelected  AND  bIWrappingChannelPiston1_Home   AND bIWrappingChannelPiston2_Home
		 AND bIWrappingChannelPiston3_Home AND NOT bAResetEnabled  AND SealingSafety   THEN
		TON_1(IN:= TRUE, PT:=T#1s , Q=> , ET=> );
		IF TON_1.Q THEN  bAConvRunning1:=FALSE; bAConvStartBit:= FALSE; step1:=step1+1; END_IF
		END_IF

	3:	 step1:=step1+1;


	4:	IF NOT bQASealingConveyorMotor AND NOT bAPauseSeq   AND (  bWCSStart1 OR bWCSStart1_24 OR bWCSStart3 OR bWCSStart3_24 ) AND SealingSafety
		AND bIWrappingCone1 AND bIWrappingCone2 AND bIWrappingCone3 THEN
		bAWrappingCone123OnAuto:=TRUE;
		bA6conesPushedTemp:=FALSE;
		WCPReadyTemp:=FALSE;
		step1:=step1+1;
		END_IF


	5:	 bWCSStart1:=FALSE; bWCSStart3:=FALSE;	step1:=step1+1;


	6:	IF bAWrappingCone123OnAuto AND bIWrappingChannelPiston1_End AND bIWrappingChannelPiston2_End AND bIWrappingChannelPiston3_End
		  AND NOT bAWrap_PistRsError AND bAFilmLoadedCom AND SealingSafety THEN
		bAConvRunning1:=FALSE;
		bAWrappingCone123FwdCom:=TRUE;
		TON_1(IN:= FALSE);
		step1:=step1+1;
		ELSIF  bAWrappingCone123OnAuto AND bIWrappingChannelPiston1_End AND bIWrappingChannelPiston2_End AND bIWrappingChannelPiston3_End
		AND NOT bAWrap_PistRsError  AND NOT bAFilmLoadedCom THEN
		bAFlimNotLoaded:=TRUE;
		bAWrappingCone123OnAuto:=FALSE;
		bAWrapConeCyl123:=FALSE;
		bAPolythinSheetError:=TRUE;
		bSheetNotFeeded:='Sheet NOT Feeded';
		step1:=step1+3;
		END_IF

	7:	  step1:=step1+1;


	8:	 IF bAWrappingCone123FwdCom AND NOT bAPauseSeq  THEN
		bAFilmLoadedCom:=FALSE;
		bAWrappingCone123OnAuto:=FALSE;
		step1:=step1+2;
		END_IF

	9:	 IF bFilmErrClear THEN bSheetNotFeeded:='Continue Machine Operation';  bAFlimNotLoaded:=FALSE;bAConvRunning1:=FALSE;  step1:=step1+1;END_IF

	10:	bAWrapConeCyl123:=FALSE;
		bA3ConeWrappOver:=TRUE;
		step1:=step1+1;

	11:	bFilmErrClear:=FALSE;step1:=step1+1;

	12:	 IF  bIWrappingChannelPiston1_Home   AND bIWrappingChannelPiston2_Home AND bIWrappingChannelPiston3_Home   THEN
		bASet1Comp:=TRUE;
		bAWrappingCone123FwdCom:=FALSE;
		bA3Pushed:=TRUE;
		bCount_ConvLockBit:=FALSE;
		step1:=0;
		END_IF
END_CASE













(*===============Wrapping Conveyor and Piston  4th and 5th Cone  Logic  in auto Mode for 2*3 model==================*)

WrapR_TRIG_3_23(CLK:=bAWrappingConvStart3_23 , Q=> );


IF WrapR_TRIG_3_23.Q THEN bAWrappingConvStartAuto3_23:=TRUE; END_IF


WrapConvStartDly3_23(IN:= bAWrappingConvStartAuto3_23, PT:=t#0.5s , Q=> , ET=> );


IF bAutoModeOn AND  WrapConvStartDly3_23.Q AND  bIWrappingChannelPiston1_Home  AND bIWrappingChannelPiston2_Home
AND bIWrappingChannelPiston3_Home AND  bAconvReayTemp AND NOT bACheckWrappConvError2 AND NOT bACheckWrappConvError3
AND NOT   bIWrappingCone1 AND NOT   bIWrappingCone2 AND NOT bIWrappingCone3  AND b2_3SetHmiSelected  THEN
bQAWrappingConveyorMotor3_23:=TRUE;
bAWrappingConvStart3_23:=FALSE;
bAWrappingConvStartAuto3_23:=FALSE;

ELSIF bAutoModeOn AND  WrapConvStartDly3_23.Q AND  bIWrappingChannelPiston1_Home  AND bIWrappingChannelPiston2_Home
AND bIWrappingChannelPiston3_Home AND  bAconvReayTemp AND (  bIWrappingCone1 OR  bIWrappingCone2 OR bIWrappingCone3 )
AND NOT bACheckWrappConvError2 (*AND NOT bACheckWrappConvError3  *) AND b2_3SetHmiSelected THEN
bACheckWrappConvError3:=TRUE;
ConeMissAlarm:='Check Wrapping Sensor 1_2_3';
END_IF

IF  bASet1Comp AND bQAWrappingConveyorMotor3_23 AND  bAutoModeOn(* AND   bIWrappingCone1*) AND bIWrappingCone2 THEN
bQAWrappingConveyorMotor3_23:=FALSE;
  (*bAWrappingConvStartAuto3_23:=FALSE;  *)  (*==========new modify on 06.10.16==============*)
  bA3Pushed:=FALSE;
bAconvReayTemp:=FALSE;
bWrapConvStopped3:=TRUE;

END_IF
(*

IF bAWrappingConvStartAuto3_23 AND NOT bCount_ConvLockBit AND bIWrappingCone1 THEN R_Bit1:=TRUE ; END_IF

IF bAWrappingConvStartAuto3_23  AND NOT bCount_ConvLockBit AND bIWrappingCone2 THEN R_Bit2:=TRUE;  END_IF

IF bAWrappingConvStartAuto3_23 AND NOT bCount_ConvLockBit  AND bIWrappingCone3 THEN R_Bit3:=TRUE; END_IF


(*===============Wrong Cone Or Sheet sensing error=====================*)
IF  R_Bit1 OR R_Bit2 OR R_Bit3  AND NOT bConeMiss2AtWrapConv  (* AND  bIWrappingChannelPiston1_Home AND bIWrappingChannelPiston2_Home AND bIWrappingChannelPiston3_Home AND *) THEN
bACheckWrappConvError3:=TRUE;
END_IF
*)

IF bACheckWrappConvError3 AND( bErrorReset OR bStopHmi ) AND b2_3SetHmiSelected AND NOT bIWrappingCone1 AND NOT bIWrappingCone2   AND NOT bIWrappingCone3 THEN bACheckWrappConvError3:=FALSE;  END_IF


(*===============Wrapping Conveyor and Piston   6th Cone  Logic  in auto Mode for 2*3 model==================*)

WrapR_TRIG_6_23(CLK:=bAWrappingConvStart4_23 , Q=> );


IF WrapR_TRIG_6_23.Q THEN bAWrappingConvStartAuto4_23:=TRUE; END_IF


WrapConvStartDly6_23(IN:= bAWrappingConvStartAuto4_23, PT:=t#0.5s , Q=> , ET=> );


IF bAutoModeOn AND  WrapConvStartDly6_23.Q AND b2_3SetHmiSelected AND   bIWrappingChannelPiston1_Home AND bIWrappingChannelPiston2_Home
AND bIWrappingChannelPiston3_Home  AND NOT bACheckWrappConvError4 AND NOT bIWrappingCone3  THEN
bQAWrappingConveyorMotor4_23:=TRUE;
bAConvRunning2:=TRUE;
bAWrappingConvStartAuto4_23:=FALSE;
ELSIF  bAutoModeOn AND  WrapConvStartDly6_23.Q AND  bIWrappingChannelPiston1_Home AND bIWrappingChannelPiston2_Home
AND bIWrappingChannelPiston3_Home  AND  bIWrappingCone3 AND b2_3SetHmiSelected  THEN
bACheckWrappConvError4:=TRUE;
ConeMissAlarm:='Check Wrapping Sensor 1_2_3';
bCone1LockBit:=TRUE;
END_IF

IF  bASet1Comp AND  bAutoModeOn AND  bQAWrappingConveyorMotor4_23  AND bAConvRunning2(* AND  bIWrappingCone1 AND bIWrappingCone2  *)
AND bIWrappingCone3 AND b2_3SetHmiSelected  THEN
bQAWrappingConveyorMotor4_23:=FALSE;
bWrapConvStopped4:=TRUE;

(*  bAWrapConeCyl123_23:=TRUE;   *)
END_IF


(*

(*===============Wrong Cone Or Sheet sensing error FOR 6TH Cone=======================*)
IF NOT bCount_ConvLockBit2 AND  bAutoModeOn AND  bAWrappingConvStartAuto4_23 AND  bIWrappingChannelPiston1_Home AND bIWrappingChannelPiston2_Home AND bIWrappingChannelPiston3_Home  AND ( bIWrappingCone1 AND bIWrappingCone2  AND bIWrappingCone3 ) THEN
bACheckWrappConvError4:=TRUE;
bCone1LockBit:=TRUE;
(*ConeMissAlarm:='Check Wrapping Sensor 1 & 2 & 3';*)
END_IF
*)
IF bACheckWrappConvError4 AND ( bErrorReset OR  bStopHmi)   AND NOT  bIWrappingCone3   THEN   bACheckWrappConvError4:=FALSE; ConeMissAlarm:='';  END_IF





(*===============Wrapping piston 123 on/off logic for  2*3 model(4 ,5,6th cone) ====================*)
CASE step5 OF

	0:	TON_2(IN:= FALSE);
		step5:=step5+1;

	1:	step5:=step5+1;

	2:	IF bAutoModeOn AND  bAWrapConeCyl123_23 AND b2_3SetHmiSelected   AND  bIWrappingChannelPiston1_Home   AND bIWrappingChannelPiston2_Home
		 AND bIWrappingChannelPiston3_Home AND NOT bAResetEnabled    THEN
		TON_2(IN:= TRUE, PT:=t#1s , Q=> , ET=> );
		IF TON_2.Q THEN  step5:=step5+1; END_IF
		END_IF

	3:	 step5:=step5+1;

	4:	IF NOT bQASealingConveyorMotor AND bWCSStart2  AND NOT bAPauseSeq AND SealingSafety AND b2_3SetHmiSelected  AND bIWrappingCone1
		AND bIWrappingCone2 AND bIWrappingCone3  THEN
		 bAWrappingCone123_23OnAuto:=TRUE;
		bAByPassOn2:=FALSE;
		 step5:=step5+1;
		END_IF

	5:	bWCSStart2:=FALSE;
		step5:=step5+1;

	6:	IF bAWrappingCone123_23OnAuto AND bIWrappingChannelPiston1_End AND bIWrappingChannelPiston2_End AND bIWrappingChannelPiston3_End
		  AND NOT bAWrap_PistRsError  AND bAFilmLoadedCom AND SealingSafety  AND b2_3SetHmiSelected THEN
		bAConvRunning2:=FALSE;
		bAWrappingCone123_23FwdCom:=TRUE;
		TON_2(IN:= FALSE);

		step5:=step5+1;
		ELSIF  bAWrappingCone123_23OnAuto AND bIWrappingChannelPiston1_End AND bIWrappingChannelPiston2_End AND bIWrappingChannelPiston3_End AND NOT bAWrap_PistRsError  AND NOT bAFilmLoadedCom THEN
		bAFlimNotLoaded:=TRUE;
		bAWrapConeCyl123_23:=FALSE;
		bAPolythinSheetError:=TRUE;
		bSheetNotFeeded:='Sheet NOT Feeded';
		step5:=step5+3;
		END_IF

	7:	 step5:=step5+1;

	8: IF bAWrappingCone123_23FwdCom   AND NOT bAPauseSeq  THEN
		bAWrappingCone123_23OnAuto:=FALSE;
		step5:=step5+2;
		END_IF

	9:	bAWrappingCone123_23OnAuto:=FALSE;
		 IF bFilmErrClear THEN bSheetNotFeeded:='Continue Machine Operation'; bAFlimNotLoaded:=FALSE;bAConvRunning2:=FALSE; step5:=step5+1;END_IF

	10:	bAWrapConeCyl123_23:=FALSE;
		bA6ConeWrappOver23:=TRUE;
		bASet1Comp:=FALSE;
		step5:=step5+1;

	11:	bFilmErrClear:=FALSE;step5:=step5+1;

	12:	 IF  bIWrappingChannelPiston1_Home   AND bIWrappingChannelPiston2_Home AND bIWrappingChannelPiston3_Home   THEN
		bAWrappingCone123_23FwdCom:=FALSE;
		bA6conesPushed:=TRUE;
		bA6conesPushedTemp:=TRUE;
		bCount_ConvLockBitTemp:=FALSE;
		step5:=0;
		END_IF
END_CASE


IF bA6conesPushed AND CounterTilt23.CV<=3 THEN
bANextLayerStarted:=TRUE;
END_IF


IF bA3Pushed OR bA6conesPushed AND bAFirstConeAtWrapConv THEN
bAConvStartInterlock:=TRUE;
ELSE
bAConvStartInterlock:=FALSE;
END_IF

(*

IF bAConvFirstStartUnitB THEN
baConveyerStarted:=TRUE;
END_IF
IF baConveyerStarted AND



*)

WrappingCone1RT(CLK:=( bIWrappingCone1 (*AND bQAWrappingConveyorMotor*) ), Q=> );



WrappingConvRT(CLK:= bQWrappingConveyorMotor , Q=> );

IF  WrappingConvRT.Q THEN
bAWrapConvStarted:=TRUE;

END_IF

IF WrappingCone1RT.Q THEN WCS1Sensed:=TRUE; END_IF

IF WCS1Sensed (*  AND bAWrapConvStarted OR bConvRunning  *)THEN
bAInterlockCountStart:=TRUE;
ELSE
bAInterlockCountStart:=FALSE;
 END_IF



IF  bQWrappingConveyorMotor AND NOT bIWrappingCone1 AND bAutoModeOn THEN
WCS1Sensed:=FALSE;
END_IF

(*

TON_6(IN:=WCS1Sensed , PT:=T#0.2s , Q=> , ET=> );

IF TON_6.Q THEN bAWrapConvStarted:=FALSE; END_IF


IF InterLockCounter.CV = 2 AND bAutoModeOn THEN
TimerStartBit:=TRUE;
bAWrapConvStarted:=FALSE;
TON_10(IN:=TimerStartBit , PT:=t#0.2s , Q=> , ET=> );

 END_IF


IF TON_10.Q AND bQWrappingConveyorMotor THEN
bConvRunning:=TRUE;
END_IF

*)

(*=============== Interlock Logic for  2*3 WCS conveyor===================*)


IF bRowStopperIntOver THEN
bSaelUnitIntOverTemp:=TRUE;
END_IF



CASE step6 OF


0:	IF bSaelUnitIntOverTemp  AND b2_3SetHmiSelected THEN                             (*========= need to check for reset Logic=    step6:=0    =======*)
	Step6:=Step6+1;
	END_IF

1:	bWCSStart1:=TRUE;
	bRowStopperIntOver:=FALSE;
	Step6:=Step6+1;

2:	IF  bASealConvEnd1 THEN
	bSaelUnitIntOverTemp:=FALSE;
	Step6:=Step6+1;
	END_IF

3:	bWCSStart2:=TRUE;
	bASealConvEnd1:=FALSE;
	Step6:=Step6+1;


4:	IF bASealConvEnd2  THEN
	Step6:=Step6+1;
	END_IF

5:	bWCSStart3:=TRUE;
	bASealConvEnd2:=FALSE;
	Step6:=2;

END_CASE


(*
(*=============== Interlock Logic for  2*4 WCS conveyor===================*)


CASE step7 OF


0:	IF bSaelUnitIntOverTemp AND b2_4SetHmiSelected  THEN                                    (*========= need to check for reset Logic=    step7:=0    =======*)
	Step7:=Step7+1;
	END_IF

1:	bWCSStart1_24:=TRUE;
	Step7:=Step7+1;

2:	IF  bASealConvEnd1_24 THEN
	bSaelUnitIntOverTemp:=FALSE;
	Step7:=Step7+1;
	END_IF

3:	bWCSStart2_24:=TRUE;
	bASealConvEnd1_24:=FALSE;
	Step7:=Step7+1;


4:	IF bASealConvEnd2_24  THEN
	Step7:=Step7+1;
	END_IF

5:	bWCSStart3_24:=TRUE;
	bASealConvEnd2_24:=FALSE;
	Step7:=2;

END_CASE

*)

IF NOT bIEmergencySwitch OR bStopHmi  OR bServoOff OR bIMcStop THEN
bAWrappingConvStartAuto3_23:=FALSE;
bAWrappingConvStartAuto4_23:=FALSE;
bAWrappingConvStart4_23:=FALSE;
bAWrappingConvStartAuto:=FALSE;
bQAWrappingConveyorMotor1:=FALSE;
bAWrappingConvStartAuto2:=FALSE;
bQAWrappingConveyorMotor2:=FALSE;
bQAWrappingConveyorMotor3:=FALSE;
bQAWrappingConveyorMotor4:=FALSE;
bQAWrappingConveyorMotor5:=FALSE;
WrapConvStartDly3_23(IN:= FALSE);
bAConvRunning1:=FALSE;
bASet1Comp:=FALSE;
bAWrappingConvStartAuto3:=FALSE;
bAWrapConeCyl3:=FALSE;
bAWrapConeCyl123:=FALSE;
WCS1Sensed:=FALSE;
bAWrappingConvStart1_23:=FALSE;
bSaelUnitIntOver:=FALSE;
bWCSStart1:=FALSE;
bWCSStart2:=FALSE;
bWCSStart3:=FALSE;
bASealConvEnd1:=FALSE;
bASealConvEnd2:=FALSE;
InterLockCounter.RESET:=TRUE;
bAWrappingCone123OnAuto:=FALSE;
bAWrappingCone123_23OnAuto:=FALSE;
bQAWrappingConveyorMotor4_23:=FALSE;
bQAWrappingConveyorMotor3_23:=FALSE;
bCount_ConvLockBit2:=FALSE;
bCount_ConvLockBit:=FALSE;
step1:=0;
step2:=0;
step3:=0;
step4:=0;
step5:=0;
step6:=0;
ELSE
InterLockCounter.RESET:=FALSE;
END_IF
END_PROGRAM

(* POU Auto1/Tilt_Piston_24, ST *)
PROGRAM Tilt_Piston_24
VAR
	CounterTiltRst: BOOL;
	step: INT;
	bATiltPistonFwdStart: BOOL;
	test1: BOOL;
	bAConeFeedingStarted: BOOL;
	bAfeedingCom: BOOL;
	bAFeedingRev: BOOL;
	NotbAFeedingRev: BOOL;
	RstStep: INT;
END_VAR
		IF bRTiltPistonReset  AND bIForwardPistonHome AND bIReversePistonHome THEN
		step:=0;
		bATiltPistonFwdStart:=FALSE;
		bAConeFeedingStarted:=FALSE;
		bAfeedingCom:=FALSE;
		bAFeedingRev:=FALSE;
		NotbAFeedingRev:=FALSE;
		bA4thConeFeedStartAuto23:=FALSE;
		bA4thConeFeedStart23:=FALSE;;
		bA6thConeFeedStartAuto23:=FALSE;
		bATiltPistonInHome:=FALSE;
		bA5thConeFeedStart:=FALSE;
		END_IF




bQAConeTiltingPistonValve1:=bATiltPistonFwdStart;


IF bQAConeFeedingPistonValve  AND NOT NotbAFeedingRev THEN bAConeFeedingStarted:=TRUE; END_IF

IF bAConeFeedingStarted AND bIConeFeedingPistonEnd  AND NOT NotbAFeedingRev THEN bAfeedingCom:=TRUE;  END_IF

IF bAfeedingCom AND NOT bIConeFeedingPistonEnd AND NOT NotbAFeedingRev THEN bAFeedingRev:=TRUE;  bAConeFeedingStarted:=FALSE;   bAfeedingCom:=FALSE;  END_IF

IF  CounterTilt.CV= 1 OR  CounterTilt.CV= 3 OR  CounterTilt.CV= 6 OR  CounterTilt.CV= 8 THEN
NotbAFeedingRev:=TRUE;
ELSE
NotbAFeedingRev:=FALSE;
END_IF

IF bATiltPistonFwdStart  AND bITiltingEnd THEN     bAFeedingRev:=FALSE; END_IF



	                                                                        (*===========Cone Tilting Piston Reset Logic===========*)

CASE step OF

	0:	IF  CounterTilt.CV=1 AND NOT bIConeFeedingPistonEnd    AND bAutoModeOn   AND bIForwardPistonHome AND bIReversePistonHome  THEN
		bATiltPistonFwdStart:=FALSE;  step:=step+1;  END_IF
		 sMessage_23_Tilting:='Check Forward and Reverse Piston Home Reed Switch';


	1:	IF NOT bAPauseSeq THEN  step:=step+1;   END_IF                                (* Cone 1 Logic  Over*)



	2:	 IF  CounterTilt.CV=2 AND   bAFeedingRev   AND bIForwardPistonHome AND bIReversePistonHome AND bIConeFeedingPistonHome  THEN
		bATiltPistonFwdStart:=TRUE;
		bATiltEnable1_24:=FALSE; step:=step+1; END_IF
		sMessage_23_Tilting:='Check Forward ,  Reverse & Cone Feeding Piston Home Reed Switch';

	3:	IF NOT bAPauseSeq THEN step:=step+1; END_IF                                   (* Cone 2 Logic  Over*)



	4:	 IF  CounterTilt.CV=3  AND bIForwardPistonHome AND bIReversePistonHome  AND bIConeFeedingPistonHome  THEN
		bATiltPistonFwdStart:=TRUE; step:=step+1;END_IF
		 sMessage_23_Tilting:='Check Forward ,  Reverse & Cone Feeding Piston Home Reed Switch';


	5:	IF NOT bAPauseSeq THEN step:=step+1; END_IF

	6:	  IF (* CounterTilt.CV=4 *) bATiltEnable2_24 AND   bIConeFeedingPistonHome AND bIForwardPistonHome AND bIReversePistonHome THEN
		bATiltPistonFwdStart:=FALSE;step:=step+1; END_IF
		sMessage_23_Tilting:='Check Forward ,  Reverse & Cone Feeding Piston Home Reed Switch';


	7:	IF NOT bAPauseSeq THEN step:=step+1; END_IF                               (* Cone 3 Logic  Over*)




	8:  IF  CounterTilt.CV= 4 AND  bAFeedingRev AND bIForwardPistonHome AND bIReversePistonHome   THEN
		bATiltPistonFwdStart:=TRUE;
		bATiltEnable2_24:=FALSE; step:=step+1; END_IF
		 sMessage_23_Tilting:='Check Forward and Reverse Piston Home Reed Switch';

	9:	IF NOT bAPauseSeq THEN step:=step+1; END_IF

	10:  IF bAtiltGoHome THEN
		bATiltPistonFwdStart:=FALSE;
		bA5thConeFeedStart:=TRUE;
		step:=step+1;
		END_IF

	11:	IF NOT bAPauseSeq THEN step:=step+1; END_IF                           (* Cone 4 Logic  Over*)




	12:	IF  CounterTilt.CV=5 AND bIConeFeedingPistonHome AND bIForwardPistonHome AND bIReversePistonHome   THEN
		bATiltPistonFwdStart:=FALSE; step:=step+1; END_IF
		sMessage_23_Tilting:='Check Forward ,  Reverse & Cone Feeding Piston Home Reed Switch';


	13:	IF NOT bAPauseSeq THEN step:=step+1; END_IF

	14:	IF CounterTilt.CV= 5 AND    bAFeedingRev AND bIForwardPistonHome AND bIReversePistonHome THEN
		bATiltPistonFwdStart:=TRUE; step:=step+1; END_IF
		 sMessage_23_Tilting:='Check Forward and Reverse Piston Home Reed Switch';

	15:	IF NOT bAPauseSeq THEN step:=step+1; END_IF

	16:	step:=step+1;

	17:	IF NOT bAPauseSeq THEN step:=step+1; END_IF                           (* Cone 5 Logic  Over*)





	18:	IF CounterTilt.CV= 6 AND bIConeFeedingPistonHome   AND bIForwardPistonHome AND bIReversePistonHome THEN
		step:=step+1; END_IF
		sMessage_23_Tilting:='Check Forward ,  Reverse & Cone Feeding Piston Home Reed Switch';

	19:	IF NOT bAPauseSeq THEN step:=step+1; END_IF

	20:	IF(* CounterTilt.CV= 7 *) bATiltEnable3_24  AND bIConeFeedingPistonHome    AND bIForwardPistonHome AND bIReversePistonHome THEN
		bATiltPistonFwdStart:=FALSE; step:=step+1; END_IF
		sMessage_23_Tilting:='Check Forward ,  Reverse & Cone Feeding Piston Home Reed Switch';


	21:	IF NOT bAPauseSeq THEN step:=step+1; END_IF                           (* Cone 6 Logic  Over*)





	22:	IF CounterTilt.CV= 7 AND bAFeedingRev    AND bIForwardPistonHome AND bIReversePistonHome THEN
		bATiltPistonFwdStart:=TRUE;
		bATiltEnable3_24:=FALSE; step:=step+1; END_IF
		 sMessage_23_Tilting:='Check Forward and Reverse Piston Home Reed Switch';

	23:	IF NOT bAPauseSeq THEN step:=step+1; END_IF

	24:	IF (* CounterTilt.CV= 1*) bATiltEnable1_24  AND bIConeFeedingPistonHome    AND bIForwardPistonHome AND bIReversePistonHome THEN
		bATiltPistonFwdStart:=FALSE; step:=0; END_IF
		sMessage_23_Tilting:='Check Forward ,  Reverse & Cone Feeding Piston Home Reed Switch';


                                                                                                                                              (* Cone 7 Logic  Over*)

END_CASE






(*
		(*===========Cone Tilting Piston On/Off Logic===========*)


		IF     bAutoModeOn AND  bConeEvenCount AND bIConeFeedingPistonEnd AND bIForwardPistonHome AND bIReversePistonHome AND NOT  bIForwardPistonEnd AND NOT  bIReversePistonEnd THEN
		bQAConeTiltingPistonValve:=TRUE;
		END_IF

		IF   bAutoModeOn AND CounterTilt.CV=4 AND  bIConeFeedingPistonHome AND bIForwardPistonHome AND bIReversePistonHome AND NOT  bIForwardPistonEnd AND NOT  bIReversePistonEnd   THEN
		bQAConeTiltingPistonValve:=FALSE;
		END_IF


*)
END_PROGRAM

(* POU Auto1/FwdRevPiston_2_4, ST *)
PROGRAM FwdRevPiston_2_4
VAR
	step: INT;
	bA2ndConeReached: BOOL;
	bA3rdConeReached: BOOL;
	bA4thConeReached: BOOL;
	bA5thConeReached: BOOL;
	bA6thConeReached: BOOL;
	bA7thConeReached: BOOL;
	bA8thConeReached: BOOL;
	fs: BOOL;
END_VAR
	                             (*=============================Forward and Reverse piston On/Off logic For 2*4 model=======================*)



CASE step OF


	 0:	 IF CounterTilt.CV=1 AND bIConeFeedingPistonEnd  THEN bAFirstConeReached:=TRUE; step:=step+1; END_IF

	 1:	 IF NOT bAPauseSeq THEN step:=step+1; END_IF

 	 2:  	IF b2_4SetHmiSelected AND NOT bQAWrappingConveyorMotor AND NOT bACheckWrappConvError5 AND
		 bAutoModeOn  AND bAFirstConeReached AND bITiltingHome AND  InterLockCounter.CV = 0 AND NOT bAPauseSeq  THEN
		bQAForwardPistonValve:=TRUE; step:=step+1; END_IF

	 3:	IF NOT bAPauseSeq THEN step:=step+1; END_IF

	 4:	IF b2_4SetHmiSelected AND bAutoModeOn AND bIForwardPistonEnd AND NOT bAPauseSeq THEN
		bA8thoneReachecdWCS:=FALSE;
		bQAForwardPistonValve:=FALSE;
		bAFirstConeReached:=FALSE;
		bAWrappingConvStart1:=TRUE;
		bAConeFeedPistonLockOk:=TRUE; step:=step+1;END_IF

	5:     IF NOT bAPauseSeq THEN step:=step+1; END_IF                                                (* Cone 1 Logic  Over*)




	6:	IF CounterTilt.CV=2 AND bIConeFeedingPistonEnd  AND NOT bAPauseSeq  THEN
		bA2ndConeReached:=TRUE;
		(*bAWrappingConvStart1:=FALSE;*) step:=step+1; END_IF

	7:	IF NOT bAPauseSeq THEN step:=step+1; END_IF                                              (* Cone 2 Logic  Over*)




	8:	IF CounterTilt.CV=3 AND bIConeFeedingPistonEnd  AND  NOT bAPauseSeq THEN
		bA3rdConeReached:=TRUE; step:=step+1; END_IF

	9:	IF NOT bAPauseSeq THEN step:=step+1; END_IF

	10:	IF b2_4SetHmiSelected AND bAutoModeOn AND NOT bACheckWrappConvError1 AND NOT bQAWrappingConveyorMotor
		AND bITiltingEnd AND bA2ndConeReached AND bA3rdConeReached AND InterLockCounter.CV=1 AND NOT bAPauseSeq  THEN
		bQAForwardPistonValve:=TRUE;
		bQAReversePistonValve:=TRUE; step:=step+1; END_IF

	11:	IF NOT bAPauseSeq THEN step:=step+1; END_IF

	12:	IF b2_4SetHmiSelected AND bAutoModeOn AND bIConeFeedingPistonHome  AND bIForwardPistonEnd AND bIReversePistonEnd AND   NOT bAPauseSeq   THEN
		bQAForwardPistonValve:=FALSE;
		bQAReversePistonValve:=FALSE;
		bA2ndConeReached:=FALSE;
		bA3rdConeReached:=FALSE;
		bAWrappingConvStart2:=TRUE;
		bATiltEnable2_24 := TRUE; step:=step+1; END_IF

	13:	IF NOT bAPauseSeq THEN step:=step+1; END_IF                                                  (* Cone 3 Logic  Over*)




                                                                     (*-=========================mod need here=======================*)
	14:	IF  CounterTilt.CV=4 AND bIConeFeedingPistonEnd THEN
		bA4thConeReached:=TRUE;
		(*bAWrappingConvStart2:=FALSE;*) step:=step+1; END_IF

	15:	IF NOT bAPauseSeq THEN step:=step+1; END_IF

	16:	IF b2_4SetHmiSelected AND bAutoModeOn AND NOT bACheckWrappConvError2 AND NOT bQAWrappingConveyorMotor
		AND  bA4thConeReached  AND bITiltingEnd AND bIReversePistonHome AND  InterLockCounter.CV=3  AND NOT bAPauseSeq  THEN
		bQAReversePistonValve:=TRUE; step:=step+1; END_IF

	17:	IF NOT bAPauseSeq THEN step:=step+1; END_IF

	18:	IF b2_4SetHmiSelected AND bAutoModeOn AND bIReversePistonEnd  AND bITiltingEnd   AND NOT bAPauseSeq THEN
		bQAReversePistonValve:=FALSE;
		bA4thConeReached:=FALSE;
		bAWrappingConvStart3:=TRUE; step:=step+1; END_IF

	19:	IF NOT bAPauseSeq THEN step:=step+1; END_IF

	20:	 IF b2_4SetHmiSelected AND bAutoModeOn AND bIReversePistonHome  AND NOT bAPauseSeq  THEN
		bAtiltGoHome:=TRUE;
		(*bAWrappingConvStart3:=FALSE;*) step:=step+1; END_IF

	21:	IF NOT bAPauseSeq THEN step:=step+1; END_IF                                                             (* Cone 4 Logic  Over*)




	22:	IF  CounterTilt.CV=5 AND bIConeFeedingPistonEnd THEN
		bA5thConeReached:=TRUE;
		bAtiltGoHome:=FALSE; step:=step+1; END_IF

	23:	IF NOT bAPauseSeq THEN step:=step+1; END_IF                                                               (* Cone 5 Logic  Over*)




	24:	IF CounterTilt.CV=6 AND bIConeFeedingPistonEnd  THEN
		bA6thConeReached:=TRUE; step:=step+1; END_IF

	25:	IF NOT bAPauseSeq THEN step:=step+1; END_IF

	26:	IF b2_4SetHmiSelected AND bAutoModeOn AND NOT bQAWrappingConveyorMotor AND NOT bACheckWrappConvError3 AND NOT bAPauseSeq
		AND  bA5thConeReached AND bA6thConeReached  AND bITiltingEnd AND bIReversePistonHome  AND bIForwardPistonHome AND  InterLockCounter.CV=4   THEN
		bQAForwardPistonValve:=TRUE;
		bQAReversePistonValve:=TRUE;step:=step+1; END_IF

	27:	IF NOT bAPauseSeq THEN step:=step+1; END_IF

	28:	IF b2_4SetHmiSelected AND bAutoModeOn AND bIConeFeedingPistonHome  AND bIForwardPistonEnd AND bIReversePistonEnd AND NOT bAPauseSeq   THEN
		bQAForwardPistonValve:=FALSE;
		bQAReversePistonValve:=FALSE;
		bA5thConeReached:=FALSE;
		bA6thConeReached:=FALSE;
		bAWrappingConvStart4:=TRUE;
		bATiltEnable3_24:=TRUE; step:=step+1; END_IF

	29:	IF NOT bAPauseSeq THEN step:=step+1; END_IF                                                          (* Cone 6 Logic  Over*)




	30:	IF  CounterTilt.CV=7 AND bIConeFeedingPistonEnd THEN
		(*bAWrappingConvStart4:=FALSE;*)
		bA7thConeReached:=TRUE; step:=step+1; END_IF

	31:	IF NOT bAPauseSeq THEN step:=step+1; END_IF                                                        (* Cone 7 Logic  Over*)




	32:	IF CounterTilt.CV=8 AND bIConeFeedingPistonEnd  THEN
		bA8thConeReached:=TRUE;step:=step+1;END_IF

	33:	IF NOT bAPauseSeq THEN step:=step+1; END_IF

	34:	IF b2_4SetHmiSelected AND bAutoModeOn AND NOT bACheckWrappConvError4 AND NOT bQAWrappingConveyorMotor   AND  bA7thConeReached
		 AND bA8thConeReached  AND bITiltingEnd AND bIReversePistonHome  AND bIForwardPistonHome AND  InterLockCounter.CV=6 AND NOT bAPauseSeq    THEN
		bQAForwardPistonValve:=TRUE;
		bQAReversePistonValve:=TRUE;step:=step+1; END_IF

	35:	IF NOT bAPauseSeq THEN step:=step+1; END_IF

	36:	IF b2_4SetHmiSelected AND bAutoModeOn AND bIConeFeedingPistonHome  AND bIForwardPistonEnd AND bIReversePistonEnd  AND NOT bAPauseSeq   THEN
		bQAForwardPistonValve:=FALSE;
		bQAReversePistonValve:=FALSE;
		bA7thConeReached:=FALSE;
		bA8thConeReached:=FALSE;
		bAWrappingConvStart5:=TRUE; step:=step+1; END_IF

	37:	IF NOT bAPauseSeq THEN step:=step+1; END_IF                                                          (* Cone 8 Logic  Over*)

	38:	 IF  bIReversePistonHome  AND bIForwardPistonHome THEN
		(*bAWrappingConvStart5:=FALSE;*)
		bATiltEnable1_24:=TRUE;
		step:=0;
		END_IF


END_CASE







IF  NOT bIEmergencySwitch OR bServoOff OR bIMcStop OR   bStopHmi  THEN
		bAWrappingConvStart5:=FALSE;
		bATiltEnable1_24:=FALSE;
		step:=0;
		bQAForwardPistonValve:=FALSE;
		bQAReversePistonValve:=FALSE;
		bA8thConeReached:=FALSE;
		bA7thConeReached:=FALSE;
		bAWrappingConvStart4:=FALSE;
		bATiltEnable3_24:=FALSE;
		bATiltEnable2_24:=FALSE;
		bA6thConeReached:=FALSE;
		bA5thConeReached:=FALSE;
		bA4thConeReached:=FALSE;
		bAtiltGoHome:=FALSE;
END_IF
END_PROGRAM

(* POU Auto1/ConeFeedPiston_24, ST *)
PROGRAM ConeFeedPiston_24
VAR
	RowStopperMotorRevDly: TON;
	RowStopperMotorRevDlyB: TON;
	iAUnitBconeFeedingcount: INT;
	bFirstCycleOver: BOOL;
	F_TRIG_1: F_TRIG;
	b8ConeDeducted: BOOL;
	b16ConeDeducted: BOOL;
	b2ndCycleOver: BOOL;
	b6ConeDeducted: BOOL;
	bFirstCycleOver2: BOOL;
	F_TRIG_2: F_TRIG;
	b12ConeDeducted: BOOL;
	b2ndCycleOver2: BOOL;
	bStartFeedConveyor: BOOL;
	UnitB_R_TRIG: R_TRIG;
	FeedConvStartTimer: BOOL;
	ton11: TON;
	ton12: TON;
	UnitbAny1ConeOK: BOOL;
	UnitBSelected: BOOL;
	Counterrst: BOOL;
	CounterTiltRst: BOOL;
	bAbove6ConeDeducted: BOOL;

	CounterTilt_Total: CTU;
	Risingok: BOOL;
	conOn: BOOL;
	test: BOOL;
	R_TRIG_1: R_TRIG;
	bQAConeFeedingPistonValve1: BOOL;
	bAConeFeedFwdStart: BOOL;
	ConeFeedConvFwdDly: TON;
	F_TRIG_3: F_TRIG;
	bAFallingTrigok: BOOL;
	bAConeFeedFwdStart2: BOOL;
	bAConeFeedFwdStart3: BOOL;
	bAConeFeedFwdStart4: BOOL;
	bAConeFeedFwdStart5: BOOL;
	step: INT;
	CounterTiltRst_R_TRIG: R_TRIG;
	bA5thConeFeedStartAuto: BOOL;
	CounterTiltEable: BOOL;
	TempBit: BOOL;
	ConeOrientationTop: TON;
	R_TRIG_3: R_TRIG;
	TON_24: TON;
	step2: INT;
	bAConeFeedingPiston_24: BOOL;
	bAConeFeedingPiston_24_2: BOOL;
	CounterTiltRst_24: BOOL;
	CounterTiltRst_24_1: BOOL;
END_VAR
IF  NOT bIEmergencySwitch OR bServoOff OR bIMcStop OR   bStopHmi  THEN
	bQAConeFeedingPistonOnAuto2:=FALSE;
	bAConeFeedFwdStart:=FALSE;
	CounterTiltRst_24:=TRUE;
	bAConeFeedPistonLockOk:=FALSE;
	 bAConeFeedingPiston_24 :=FALSE;
	bAConeFeedingPiston_24_2:=FALSE;
	TON_24(IN:= FALSE);
	bAFeedingConvOff_1:=FALSE;
	bA5thConeFeedStartAuto:=FALSE;
	step:=0;
	step2:=0;
	ELSE
	CounterTiltRst_24:=FALSE;
	END_IF



                                                                               (*======================Cone Feeding Piston On/Off  Logic for 2*4 Group ===============*)


		IF   b2_4SetHmiSelected AND bAutoModeOn AND ConeFeedConvFwdDly.Q  AND bIConeFeedingPistonHome   AND  NOT bQAFeedingConveyorMotor

		(*	AND bITiltingHome  *) AND bIForwardPistonHome AND bIReversePistonHome     AND NOT bAPauseSeq      THEN
		bQAConeFeedingPistonOnAuto2:=TRUE;
		END_IF

		IF   b2_4SetHmiSelected AND  bQAConeFeedingPistonValve AND bAutoModeOn AND  bIConeFeedingPistonEnd AND NOT bAPauseSeq  THEN
		bQAConeFeedingPistonOnAuto2:=FALSE;
		END_IF
(*

		IF  b2_4SetHmiSelected AND bAutoModeOn AND ( CounterTilt.CV=3 OR  CounterTilt.CV =5 ) AND bIConeOrientationTop AND
			bITiltingEnd AND bIForwardPistonHome AND bIReversePistonHome              THEN
		bQAConeFeedingPistonValve1:=TRUE;
		END_IF


*)
R_TRIG_1(CLK:=bQAFeedingConveyorMotor , Q=> );
IF R_TRIG_1.Q THEN ;  END_IF


IF bIConeOrientationTop  AND  b2_4SetHmiSelected  AND bQAFeedingConveyorMotor AND bIConeFeedingPistonHome  THEN

    	CounterTiltEable:=TRUE;
ELSE
	CounterTiltEable:=FALSE;
END_IF

CounterTilt(
	CU:= bAConeFeedingPiston_24,
	RESET:=(CounterTiltRst_24 OR CounterTiltRst_24_1),
	PV:=8 ,
	Q=> ,
	CV=> );


F_TRIG_3(CLK:= bIConeOrientationTop , Q=> );

IF   F_TRIG_3.Q THEN bAFallingTrigok:=TRUE; END_IF

CounterTilt_Total(
	CU:= F_TRIG_1.Q,
	RESET:= ,
	PV:= ,
	Q=> ,
	CV=> );

(*===========Cone crossing sensor single sensing logic  UnitA side======================*)


CASE step2 OF

	0:	R_TRIG_3(CLK:=CounterTiltEable , Q=> );
		IF R_TRIG_3.Q THEN TON_24(IN:= FALSE); step2:=step2+1; END_IF


	1:	bAFeedingConvOff_1:=TRUE;TON_24(IN:= FALSE);
		step2:=step2+1;


	2:	IF NOT bAPauseSeq THEN   bAConeFeedingPiston_24 :=TRUE;
		 step2:=Step2+1;END_IF

	3:	 step2:=step2+1;

	4: 	TON_24(IN :=  TRUE  , PT:=t#1.3s , Q=> , ET=> );
		IF TON_24.Q THEN  step2:=step2+1; END_IF


	5:	 step2:=step2+1;

	6:	bAConeFeedingPiston_24_2:=TRUE;
		TON_24(IN:= FALSE);
		step2:=step2+1;

	7:	 step2:=step2+1;

	8:	IF bAConeFeedingPiston_24_2 THEN bAConeFeedingPiston_24:=FALSE; step2:=step2+1; END_IF

	9:	IF NOT bAPauseSeq THEN bAConeFeedingPiston_24_2:=FALSE;
		 step2:=step2+1; END_IF

	10:  IF bIConeFeedingPistonEnd THEN
		step2:=Step2+1; END_IF

	11:	 IF bIConeFeedingPistonHome THEN bAFeedingConvOff_1:=FALSE; step2:=0; END_IF

END_CASE



                                                                        (*======================Cone Feeding Piston On/Off  Logic for 2*4 Group ===============*)


F_TRIG_2(CLK:= bIConeOrientationTop , Q=> );


CASE step OF

	0:	IF  CounterTilt.CV=1  AND bIForwardPistonHome AND b2_4SetHmiSelected AND bIReversePistonHome  AND bITiltingHome  AND NOT bAResetEnabled THEN
		bAConeFeedFwdStart:=TRUE;
		CounterTiltRst:=FALSE;
		step:=step+1; END_IF sMessage_24:='Check Forward ,Reverse & Tilting Piston Home';


	1:	IF NOT bAPauseSeq THEN step:=step+1; END_IF


	2:	 IF bIConeFeedingPistonEnd  AND b2_4SetHmiSelected THEN
		bAConeFeedFwdStart:=FALSE;
		step:=step+1; END_IF


	3:	IF NOT bAPauseSeq THEN step:=step+1; END_IF                             (* Cone 1  Logic Over *)


	4:	IF   CounterTilt.CV = 2  AND bIForwardPistonHome AND bIReversePistonHome AND bAConeFeedPistonLockOk   AND bITiltingHome  AND b2_4SetHmiSelected THEN
		 bAConeFeedFwdStart:=TRUE ;
		IF NOT bIConeFeedingPistonHome THEN step:=step+1; END_IF
		END_IF sMessage_24:='Check Forward ,Reverse & Tilting Piston Home';


	5:	IF NOT bAPauseSeq THEN step:=step+1; END_IF


	6:      IF bIConeFeedingPistonEnd AND b2_4SetHmiSelected THEN
		bAConeFeedFwdStart:=FALSE;
		bAConeFeedPistonLockOk:=FALSE; step:=step+1; END_IF

	7:	IF NOT bAPauseSeq THEN step:=step+1; END_IF                              (* Cone 2  Logic Over *)


	8:     IF  CounterTilt.CV = 3 AND bIForwardPistonHome AND bIReversePistonHome AND bITiltingEnd AND b2_4SetHmiSelected  THEN
		bAConeFeedFwdStart:=TRUE; step:=step+1; END_IF sMessage_24:='Check Forward ,Reverse & Tilting Piston Home';


	9:	IF NOT bAPauseSeq THEN step:=step+1; END_IF


	10:	 IF bIConeFeedingPistonEnd AND b2_4SetHmiSelected  THEN bAConeFeedFwdStart:=FALSE;step:=step+1; END_IF


	11:	IF NOT bAPauseSeq THEN step:=step+1; END_IF                           (* Cone 3   Logic Over *)


	12:	IF CounterTilt.CV = 4 AND bIForwardPistonHome AND bIReversePistonHome   AND bITiltingHome  AND b2_4SetHmiSelected THEN
		bAConeFeedFwdStart:=TRUE;step:=step+1; END_IF sMessage_24:='Check Forward ,Reverse & Tilting Piston Home';


	13:	IF NOT bAPauseSeq THEN step:=step+1; END_IF


	14:	IF bIConeFeedingPistonEnd AND b2_4SetHmiSelected  THEN
		bAConeFeedFwdStart:=FALSE; step:=step+1; END_IF


	15:	IF NOT bAPauseSeq THEN step:=step+1; END_IF                            (* Cone 4   Logic Over *)


	16:	IF   CounterTilt.CV = 5  AND bIForwardPistonHome AND bIReversePistonHome  AND bA5thConeFeedStartAuto  AND b2_4SetHmiSelected  THEN
		bAConeFeedFwdStart:=TRUE; step:=step+1; END_IF sMessage_24:='Check Forward ,Reverse & Tilting Piston Home';


	17:	IF NOT bAPauseSeq THEN step:=step+1; END_IF


	18:	IF bIConeFeedingPistonEnd  AND b2_4SetHmiSelected  THEN
		bAConeFeedFwdStart:=FALSE;
		bA5thConeFeedStart:=FALSE;
		bA5thConeFeedStartAuto:=FALSE; step:=step+1; END_IF


	19:	IF NOT bAPauseSeq THEN step:=step+1; END_IF                             (* Cone 5  Logic Over *)



	20: IF   CounterTilt.CV = 6  AND bIForwardPistonHome AND bIReversePistonHome AND bITiltingEnd AND b2_4SetHmiSelected  THEN
		bAConeFeedFwdStart:=TRUE;	step:=step+1; END_IF


	21:	IF NOT bAPauseSeq THEN step:=step+1; END_IF


	22:	IF bIConeFeedingPistonEnd AND b2_4SetHmiSelected THEN
		bAConeFeedFwdStart:=FALSE; step:=step+1; END_IF


	23:	IF NOT bAPauseSeq THEN step:=step+1; END_IF                               (* Cone 6  Logic Over *)


	24:	IF   CounterTilt.CV = 7  AND bIForwardPistonHome AND bIReversePistonHome   AND bITiltingHome AND b2_4SetHmiSelected  THEN
		bAConeFeedFwdStart:=TRUE; step:=step+1; END_IF sMessage_24:='Check Forward ,Reverse & Tilting Piston Home';


	25:	IF NOT bAPauseSeq THEN step:=step+1; END_IF


	26:	IF bIConeFeedingPistonEnd  AND b2_4SetHmiSelected   THEN
		bAConeFeedFwdStart:=FALSE; step:=step+1; END_IF

	27:	IF NOT bAPauseSeq THEN step:=step+1; END_IF                                  (* Cone 7  Logic Over *)



	28:	IF   CounterTilt.CV = 8  AND bIForwardPistonHome AND bIReversePistonHome  AND  bITiltingEnd AND b2_4SetHmiSelected  THEN
		bAConeFeedFwdStart:=TRUE; step:=step+1;END_IF


	29:	IF NOT bAPauseSeq THEN step:=step+1; END_IF


	30:	IF bIConeFeedingPistonEnd  AND b2_4SetHmiSelected  THEN
		bAConeFeedFwdStart:=FALSE;
		 step:=step+1; END_IF

	31:	CounterTiltRst_24_1:=TRUE; step:=step+1;

	32:	IF NOT bAPauseSeq THEN step:=step+1; END_IF                                 (* Cone 8  Logic  Over*)


	33:	CounterTiltRst_24_1:=FALSE;
		step:=0;



END_CASE



CounterTiltRst_R_TRIG(CLK:= CounterTiltRst_24, Q=> );


CounterTilt.RESET:=CounterTiltRst_R_TRIG.Q;

                                                                       (*========= This satement used to bring the cone feeding piston after 4th cone complete==========*)

		IF bA5thConeFeedStart AND bITiltingHome THEN   bA5thConeFeedStartAuto:=TRUE; END_IF

ConeFeedConvFwdDly(IN:=bAConeFeedFwdStart , PT:=t#1s , Q=> , ET=> );




IF bAResetHmi THEN
	bAConeFeedFwdStart:=FALSE;
	step:=0;
	CounterTiltRst:=FALSE;

	END_IF
END_PROGRAM

(* POU Auto/Wrapping_Unit_24, ST *)
PROGRAM Wrapping_Unit_24
VAR

	step1: INT;

	R_TRIG_1: R_TRIG;
	Counter1: CTU;
	WrapConvStartDly: TON;
	WrapR_TRIG_1: R_TRIG;
	bAWrappingConvStartAuto2: BOOL;
	WrapR_TRIG_2: R_TRIG;
	WrapConvStartDly2: TON;
	WrapR_TRIG_3: R_TRIG;
	WrapConvStartDly3: TON;
	bAWrappingConvStartAuto3: BOOL;
	WrapR_TRIG_4: R_TRIG;
	bAWrappingConvStartAuto4: BOOL;
	WrapConvStartDly4: TON;
	WrapR_TRIG_5: R_TRIG;
	bAWrappingConvStartAuto5: BOOL;
	WrapConvStartDly5: TON;
	bAWrapConeCyl1: BOOL;
	bAWrapConeCyl3: BOOL;
	bAWrapConeCyl23: BOOL;
	bASet1Comp: BOOL;
	bASet2Comp: BOOL;
	bASet: BOOL;
	bASet3Comp: BOOL;
	bA3ConeWrapStarted: BOOL;
	bA6thConeWrapStarted: BOOL;
	bA1ConeWrappOver: BOOL;
	bA2ConeWrappOver: BOOL;
	bAll3ConeWrapOver: BOOL;
	bA5ConeWrappOver: BOOL;
	bA6ConeWrappOver: BOOL;
	bA56ConeWrapOver: BOOL;
	bAWrapConeCyl23_1: BOOL;

	bATemp: BOOL;
	baConv2ndStart: BOOL;
	baConv3rdStart: BOOL;
	baConv4thStart: BOOL;
	baConv5thStart: BOOL;
	bASensorMonitorBit1: BOOL;
	bAWrappingCone123FwdCom: BOOL;
	ni: BOOL;
	step2: INT;
	bAWrappingCone3FwdCom: BOOL;
	step3: INT;
	bAWrappingCone23FwdCom: BOOL;
	step4: INT;
	bAWrappingCone23FwdCom1: BOOL;
	bASet4Comp: BOOL;

	bAWrappingConvStartAuto3_23: BOOL;
	WrapConvStartDly3_23: TON;
	bAWrapConeCyl23_1_23: BOOL;
	bAWrappingCone23_23FwdCom1: BOOL;
	WrapR_TRIG_6_23: R_TRIG;
	bAWrappingConvStartAuto4_23: BOOL;
	WrapConvStartDly6_23: TON;
	bIWrappingCone: BOOL;

	bAWrappingCone123_23FwdCom: BOOL;

	step5: INT;
	bAConvRunning1: BOOL;
	bAConvRunning2: BOOL;
	TON_1: TON;
	TON_2: TON;
	bANextLayerStarted: BOOL;
	bAConvStartInterlock: BOOL;
	bAFirstConeAtWrapConv: BOOL;
	baConveyerStarted: BOOL;
	RtrigBit1: BOOL;
	R_TRIG_3: R_TRIG;
	bASensorNok: BOOL;
	WrapConvStartDlyOver: BOOL;
	test: R_TRIG;
	WrappingCone1RT: R_TRIG;
	WrappingConvRT: R_TRIG;
	WCS1Sensed: BOOL;
	TON_3: TON;
	WCS1SenseRst1: BOOL;
	TON_6: TON;
	TON_7: TON;
	TON_8: TON;
	TON_9: TON;
	TON_10: TON;
	TimerStartBit: BOOL;
	bConvRunning: BOOL;
	test1THEN: BOOL;
	test1: BOOL;
	bSaelUnitIntOverTemp: BOOL;
	step6: INT;
	step7: INT;
	bWCSStart3_24: BOOL;
	bStopHmitemp: BOOL;
	bWCSHomeSenOk: BOOL;
	WCSCylsHomeRsErrChk: RS_Error;
	WCSCylsHomeRsErr: BOOL;
	WCSCylsEndRsErrChk: RS_Error;
	bWCSHomeEndOk: BOOL;
	WCSCylsEndRsErr: BOOL;
	WCSSensorErrChk: RS_Error;
	bAWrappingConvStartAuto3_23temp: BOOL;
	bAWrappingConvStartAuto3_23temp2: BOOL;
	R_Bit1: BOOL;
	R_Bit2: BOOL;
	R_Bit3: BOOL;
	test2: BOOL;
	R_TRIG_2: R_TRIG;
	WCPReadyTemp: BOOL;
	bWrongSenChkBit: BOOL;
	bAWrapConeCyl23_24: BOOL;
	bAWrapConeCyl23_24_1: BOOL;
	bASensorMonitorBit2: BOOL;
	bASensorMonitorBit3: BOOL;
	bAFlimNotLoaded1: BOOL;
	bAFlimNotLoaded2: BOOL;
	bAFlimNotLoaded3: BOOL;
	TR: BOOL;
	WrapR_TRIG_24_3: R_TRIG;
	WrapR_TRIG_24: R_TRIG;
END_VAR
					            (*========================Wrapping Conveyor Logic in auto Mode=================*)

bQAWrappingConveyorMotor:= (bQAWrappingConveyorMotor1 OR bQAWrappingConveyorMotor2 OR bQAWrappingConveyorMotor3 OR bQAWrappingConveyorMotor4 OR bQAWrappingConveyorMotor5 OR bQAWrappingConveyorMotor3_23 OR bQAWrappingConveyorMotor4_23 );

                                          (*========================Wrapping Conveyor  Logic for First Cone in auto Mode for 2*4 model=================*)

IF  (bAWrappingConvStart1 OR bAWrappingConvStart1_23) AND b2_4SetHmiSelected THEN RtrigBit1:=TRUE; ELSE  RtrigBit1:=FALSE;  END_IF
WrapR_TRIG_1(CLK:= RtrigBit1 , Q=> );
IF bAutoModeOn AND  WrapR_TRIG_1.Q (* OR R_TRIG_3.Q *) THEN  bAWrappingConvStartAuto:=TRUE; END_IF
WrapConvStartDly(IN:= bAWrappingConvStartAuto, PT:=t#0.5s , Q=> , ET=> );



IF bAutoModeOn AND  WrapConvStartDly.Q   AND bIWrappingChannelPiston1_Home AND bIWrappingChannelPiston2_Home AND b2_4SetHmiSelected

AND bIWrappingChannelPiston3_Home  AND WCPReady AND NOT bIWrappingCone1 AND NOT bIWrappingCone2 AND NOT bIWrappingCone3

AND NOT bACheckWrappConvError1 AND NOT bACheckWrappConvError4  AND NOT bAFlimNotLoaded3  AND NOT bAConeMissErrorAtWrpConvTemp5_24

AND NOT bWrapConvStopped4_24 THEN
bQAWrappingConveyorMotor1:=TRUE;
bAconvReayTemp2:=FALSE;
bAconvReadyTemp5:=FALSE;
InterLockCounter.RESET:=FALSE;
bAWrappingConvStartAuto:=FALSE;
bAWrappingConvStart1_23:=FALSE;
bACheckWrappConvError1:=FALSE;
bAWrappingConvStart1:=FALSE;
bAConvStartBit:=TRUE;

ELSIF bAutoModeOn AND b2_4SetHmiSelected AND  WrapConvStartDly.Q   AND bIWrappingChannelPiston1_Home AND bIWrappingChannelPiston2_Home AND NOT bQAWrappingConveyorMotor1
 AND bIWrappingChannelPiston3_Home (* AND bWrongSenChkBit *)AND (  bIWrappingCone1 OR  bIWrappingCone2 OR  bIWrappingCone3 ) AND NOT bAPauseSeq
AND NOT bACheckWrappConvError4 AND NOT bAFlimNotLoaded3  AND NOT bAConeMissErrorAtWrpConvTemp5_24 AND NOT bWrapConvStopped4_24
AND NOT bASet3Comp THEN
bACheckWrappConvError1:=TRUE;
END_IF


IF bACheckWrappConvError1 AND(  bErrorReset OR  bStopHmi ) AND b2_4SetHmiSelected THEN  bACheckWrappConvError1:=FALSE; ConeMissAlarm:=''; END_IF
R_TRIG_2(CLK:=bWrpConvIntOver , Q=> );
IF R_TRIG_2.Q THEN WCPReadyTemp:=TRUE; END_IF

IF WCPReadyTemp OR bA6conesPushedTemp THEN bWrongSenChkBit:=TRUE; ELSE  bWrongSenChkBit:=FALSE; END_IF


IF   bAutoModeOn AND  bIWrappingCone1 AND bAConvStartBit   AND b2_4SetHmiSelected THEN
 bQAWrappingConveyorMotor1:=FALSE; END_IF




				     (*===============Wrapping Conveyor 2nd and 3rd Cone  Logic  in auto Mode for 2*4  model==================*)


WrapR_TRIG_2(CLK:= ( bAWrappingConvStart2 OR bAWrappingConvStart2_23) , Q=> );

IF bAutoModeOn AND  WrapR_TRIG_2.Q THEN  bAWrappingConvStartAuto2:=TRUE; END_IF

WrapConvStartDly2(IN:= bAWrappingConvStartAuto2, PT:=t#0.5s , Q=> , ET=> );


IF bAutoModeOn AND b2_4SetHmiSelected AND  WrapConvStartDly2.Q  AND bIWrappingChannelPiston1_Home AND bIWrappingChannelPiston2_Home AND bIWrappingChannelPiston3_Home
 AND NOT bIWrappingCone2 AND NOT bIWrappingCone3  AND NOT bACheckWrappConvError2 AND NOT bAFlimNotLoaded3 THEN
	bQAWrappingConveyorMotor2:=TRUE;
	bAWrappingConvStartAuto2:=FALSE;
	bAConvRunning1:=TRUE;
	bACheckWrappConvError2:=FALSE;
	bAWrappingConvStart2:=FALSE;

ELSIF bAutoModeOn AND b2_4SetHmiSelected AND   WrapConvStartDly2.Q  AND NOT bQAWrappingConveyorMotor2 AND bIWrappingChannelPiston1_Home AND bIWrappingChannelPiston2_Home AND bIWrappingChannelPiston3_Home
 AND ( bIWrappingCone2 OR  bIWrappingCone3 )  AND NOT bAFlimNotLoaded3  AND NOT bACheckWrappConvError2 AND NOT bAPauseSeq   THEN
	bACheckWrappConvError2:=TRUE;
END_IF

IF bACheckWrappConvError2 AND (bErrorReset  OR  bStopHmi) AND b2_4SetHmiSelected  THEN bACheckWrappConvError2:=FALSE; ConeMissAlarm:='';  END_IF

IF  bAutoModeOn AND bAConvRunning1 AND bIWrappingCone3 AND b2_4SetHmiSelected  THEN
	bQAWrappingConveyorMotor2:=FALSE;
	bWrapConvStopped2:=TRUE;
 	bAWrapConeCyl123:=TRUE;


END_IF


                                                                   (*===============Wrapping Conveyor and Piston 4th Cone  Logic  in auto Mode for 2*4 model==================*)



WrapR_TRIG_24(CLK:=bAWrappingConvStart3 , Q=> );

IF bAutoModeOn AND  WrapR_TRIG_24.Q THEN bAWrappingConvStartAuto3:=TRUE; END_IF

WrapConvStartDly3(IN:= bAWrappingConvStartAuto3, PT:=t#0.5s , Q=> , ET=> );


IF bASet1Comp AND b2_4SetHmiSelected AND  bAutoModeOn AND WrapConvStartDly3.Q AND bIWrappingChannelPiston1_Home AND bIWrappingChannelPiston2_Home
AND bIWrappingChannelPiston3_Home AND NOT bIWrappingCone3 AND NOT bIWrappingCone1 AND NOT bIWrappingCone2  AND bAconvReayTemp AND NOT bAFlimNotLoaded  AND NOT bACheckWrappConvError3 THEN
	bQAWrappingConveyorMotor3:=TRUE;
	bASensorMonitorBit1:=TRUE;
	bACheckWrappConvError3:=FALSE;
	bAWrappingConvStart3:=FALSE;
ELSIF  bASet1Comp AND b2_4SetHmiSelected AND   bAutoModeOn AND WrapConvStartDly3.Q AND bIWrappingChannelPiston1_Home AND bIWrappingChannelPiston2_Home AND NOT bQAWrappingConveyorMotor3
AND bIWrappingChannelPiston3_Home AND (  bIWrappingCone1 OR  bIWrappingCone2 OR  bIWrappingCone3 ) AND bAconvReayTemp AND NOT bAFlimNotLoaded
AND NOT bACheckWrappConvError3 AND NOT bAPauseSeq  THEN
bACheckWrappConvError3:=TRUE;
END_IF

IF bACheckWrappConvError3 AND (bErrorReset  OR  bStopHmi) AND b2_4SetHmiSelected   THEN bACheckWrappConvError3:=FALSE; ConeMissAlarm:='';  END_IF

IF b2_4SetHmiSelected THEN
IF bASet1Comp AND  bAutoModeOn AND   bIWrappingCone3 AND bASensorMonitorBit1 AND b2_4SetHmiSelected  THEN
	bQAWrappingConveyorMotor3:=FALSE;
	bAWrappingConvStartAuto3:=FALSE;
	bAWrapConeCyl3:=TRUE;
	bA3Pushed:=FALSE;
	bAconvReayTemp:=FALSE;
	bWrapConvStopped4_24exp:=TRUE;
END_IF
END_IF



                                                           (*===============Wrapping Conveyor and Piston 5th and 6th Cone  Logic  in auto Mode  for 2*4 model==================*)



	WrapR_TRIG_4(CLK:=bAWrappingConvStart4 , Q=> );

IF  bAutoModeOn AND WrapR_TRIG_4.Q THEN bASensorMonitorBit1:= FALSE;  bAWrappingConvStartAuto4:=TRUE; END_IF

	WrapConvStartDly4(IN:= bAWrappingConvStartAuto4, PT:=t#0.5s , Q=> , ET=> );

IF bASet2Comp AND bAutoModeOn AND b2_4SetHmiSelected AND   WrapConvStartDly4.Q AND bIWrappingChannelPiston1_Home AND bIWrappingChannelPiston2_Home
 AND bIWrappingChannelPiston3_Home AND bAconvReadyTemp3 AND NOT bACheckWrappConvError4 AND NOT bIWrappingCone1 AND NOT  bIWrappingCone2 AND NOT  bIWrappingCone3
AND NOT bAFlimNotLoaded1  THEN
	bQAWrappingConveyorMotor4:=TRUE;
	bASensorMonitorBit2:=TRUE;
	bACheckWrappConvError4:=FALSE;
	bAWrappingConvStart4:=FALSE;
ELSIF  bASet2Comp AND bAutoModeOn AND b2_4SetHmiSelected  AND  WrapConvStartDly4.Q AND NOT bQAWrappingConveyorMotor4 AND bIWrappingChannelPiston1_Home AND bIWrappingChannelPiston2_Home
AND bIWrappingChannelPiston3_Home AND bAconvReadyTemp3  AND(  bIWrappingCone1 OR  bIWrappingCone2 OR  bIWrappingCone3 ) AND NOT bAFlimNotLoaded1
 AND NOT bACheckWrappConvError4 AND NOT bAPauseSeq   THEN
bACheckWrappConvError4:=TRUE;
END_IF

IF bACheckWrappConvError4 AND (bErrorReset  OR  bStopHmi) AND b2_4SetHmiSelected  THEN bACheckWrappConvError4:=FALSE; ConeMissAlarm:='';  END_IF

IF b2_4SetHmiSelected THEN
IF bASet2Comp AND  bAutoModeOn  AND bIWrappingCone3 AND bASensorMonitorBit2  AND b2_4SetHmiSelected THEN
	bQAWrappingConveyorMotor4:=FALSE;
	bAWrappingConvStartAuto4:=FALSE;
	bAWrapConeCyl23_24_1:=TRUE;
	b4thConePushed:=FALSE;
	bAconvReadyTemp3:=FALSE;
	bWrapConvStopped3_24:=TRUE;
END_IF
END_IF

	WrapR_TRIG_24_3(CLK:=bIWrappingCone3 , Q=> );



                                                       (*===============Wrapping Conveyor and Piston  7th and 8th Cone  Logic  in auto Mode  for 2*4 model==================*)


	WrapR_TRIG_5(CLK:=bAWrappingConvStart5 , Q=> );

IF bAutoModeOn AND WrapR_TRIG_5.Q THEN bAWrappingConvStartAuto5:=TRUE; bASensorMonitorBit2:=FALSE; END_IF

	WrapConvStartDly5(IN:= bAWrappingConvStartAuto5, PT:=t#0.5s , Q=> , ET=> );


IF bASet3Comp AND bAutoModeOn AND b2_4SetHmiSelected AND  WrapConvStartDly5.Q AND  bIWrappingChannelPiston1_Home AND bIWrappingChannelPiston2_Home
AND bIWrappingChannelPiston3_Home  AND bAconvReadyTemp4   AND NOT bIWrappingCone2 AND  NOT  bIWrappingCone3 AND NOT  bIWrappingCone1 AND NOT bAFlimNotLoaded2
AND NOT bACheckWrappConvError5 THEN
bQAWrappingConveyorMotor5:=TRUE;
bASensorMonitorBit3:=TRUE;
bACheckWrappConvError5:=FALSE;
bAWrappingConvStart5:=FALSE;
ELSIF  bASet3Comp AND bAutoModeOn  AND b2_4SetHmiSelected AND  WrapConvStartDly5.Q AND NOT bQAWrappingConveyorMotor5 AND  bIWrappingChannelPiston1_Home AND bIWrappingChannelPiston2_Home
AND bIWrappingChannelPiston3_Home  AND bAconvReadyTemp4   AND(  bIWrappingCone1 OR  bIWrappingCone2 OR  bIWrappingCone3 ) AND NOT bAFlimNotLoaded2
AND NOT bACheckWrappConvError5 AND NOT bAPauseSeq   THEN
bACheckWrappConvError5:=TRUE;
END_IF

IF bACheckWrappConvError5 AND (bErrorReset  OR  bStopHmi)  AND b2_4SetHmiSelected  THEN bACheckWrappConvError5:=FALSE; ConeMissAlarm:='';  END_IF

IF b2_4SetHmiSelected THEN
IF  bASet3Comp AND  bAutoModeOn  AND  bIWrappingCone3 AND bASensorMonitorBit3   THEN
	bQAWrappingConveyorMotor5:=FALSE;
	bAWrappingConvStartAuto5:=FALSE;
	bAWrapConeCyl23_24:=TRUE;
	b6thConePushed_24:=FALSE;
	bAconvReadyTemp4:=FALSE;
	bWrapConvStopped4_24:=TRUE;
END_IF
END_IF



                                                                                          (*===================Wrapping Pinston On/Off Logic In Auto Mode==================*)


bQAWrappingChannelPistonValve1:= (bAWrappingCone123OnAuto OR bAWrappingCone123_23OnAuto);

bQAWrappingChannelPistonValve2:=( bAWrappingCone123OnAuto OR bAWrappingCone23OnAuto OR bAWrappingCone23OnAuto1 OR bAWrappingCone123_23OnAuto );

bQAWrappingChannelPistonValve3:=( bAWrappingCone123OnAuto OR bAWrappingCone23OnAuto OR bAWrappingCone23OnAuto1 OR  bAWrappingCone3OnAuto OR bAWrappingCone123_23OnAuto  );





                                                           (*===============Wrapping piston 1 & 2nd and 3rd  Logic for Cones in auto Mode  for 2*4 model==================*)


CASE step1 OF

	0:	TON_1(IN:= FALSE); step1:=step1+1;

	1:	step1:=step1+1;

	2:	IF bAutoModeOn AND  bAWrapConeCyl123  AND NOT bACheckWrappConvError1 AND NOT  bACheckWrappConvError2 AND b2_4SetHmiSelected
		 AND NOT bAFlimNotLoaded3 AND NOT bA8thConeWrappOver AND NOT bAConeMissErrorAtWrpConvTemp1_24 AND NOT bAConeMissErrorAtWrpConvTemp2_24
		 AND SealingSafety  AND   bIWrappingChannelPiston1_Home   AND bIWrappingChannelPiston2_Home AND bIWrappingChannelPiston3_Home
		 AND NOT bAResetEnabled    THEN
		TON_1(IN:= TRUE, PT:=T#1s , Q=> , ET=> );
		 sMessage_Wrapping:='Check Wrapping Piston Home 1 & 2 & 3 Reed Switch';

		IF TON_1.Q THEN  bAConvRunning1:=FALSE; SealingOver1:=FALSE;SealingSafety:=FALSE;bASet4Comp:=FALSE;
		bAConvStartBit:=FALSE; step1:=step1+1; END_IF
		END_IF

	3:	 step1:=step1+1;


	4:	IF NOT bQASealingConveyorMotor AND NOT bACheckWrappConvError1  (*AND NOT bQSealBitAlert_24 *)AND NOT bQSealBitAlert AND b2_4SetHmiSelected
		  AND NOT bAPauseSeq AND (  bWCSStart1 OR bWCSStart1_24 OR bWCSStart3 OR bWCSStart3_24 ) AND  bIWrappingCone1 AND bIWrappingCone2
		AND bIWrappingCone3 AND NOT bAConeMissErrorAtWrpConvTemp1_24  AND NOT bAConeMissErrorAtWrpConvTemp2_24 AND NOT SealConeMissAlet_24
		AND SealingSafety  THEN
		bAWrappingCone123OnAuto:=TRUE;
		bA6conesPushedTemp:=FALSE;
		WCPReadyTemp:=FALSE; step1:=step1+1; END_IF


	5:	 bWCSStart1:=FALSE; bWCSStart3:=FALSE; step1:=step1+1;


	6:	IF bAWrappingCone123OnAuto AND bIWrappingChannelPiston1_End AND bIWrappingChannelPiston2_End AND bIWrappingChannelPiston3_End

		AND NOT bAWrap_PistRsError AND bAFilmLoadedCom  AND NOT bAConeMissErrorAtWrpConvTemp2_24  AND NOT bAConeMissErrorAtWrpConvTemp3_24
		 AND NOT bAConeMissErrorAtWrpConvTemp4_24  AND NOT bAConeMissErrorAtWrpConvTemp5_24 AND NOT bQSealBitAlert (*AND NOT bQSealBitAlert_24*)
		 AND NOT SealConeMissAlet_24 THEN
		bAConvRunning1:=FALSE;
		bAWrappingCone123FwdCom:=TRUE;
		bWrapConvStopped1_24exp:=TRUE;
		bAConeMissErrorAtWrpConvTemp2_24:=FALSE;
		TON_4_24(IN:=FALSE);
		TON_12_24(in:=FALSE);
		bWrapConvStopped2:=FALSE;
		bAConeMissErrorAtWrpConvTemp1_24:=FALSE;
 		TON_3(IN:=FALSE);
		TON_13_24(in:=FALSE);
		TON_1(IN:= FALSE); step1:=step1+1;
		ELSIF  bAWrappingCone123OnAuto AND bIWrappingChannelPiston1_End AND bIWrappingChannelPiston2_End AND bIWrappingChannelPiston3_End
		AND NOT bAWrap_PistRsError  AND NOT bAFilmLoadedCom AND NOT bAPauseSeq THEN
		bAFlimNotLoaded:=TRUE;
		bAWrappingCone123OnAuto:=FALSE;
		bAWrapConeCyl123:=FALSE;
		bAPolythinSheetError:=TRUE;
		bAConeMissErrorAtWrpConvTemp1_24:=FALSE;
 		TON_3(IN:=FALSE);
		TON_13_24(in:=FALSE);
		bAConeMissErrorAtWrpConvTemp2_24:=FALSE;
		bWrapConvStopped2:=FALSE;
 		TON_4_24(IN:=FALSE);
		TON_12_24(in:=FALSE);
		bSheetNotFeeded:='Sheet NOT Feeded'; step1:=step1+3; END_IF

	7:	  IF NOT bAPauseSeq  THEN step1:=step1+1; END_IF


	8:	 IF bAWrappingCone123FwdCom AND NOT bAPauseSeq  THEN
		bAFilmLoadedCom:=FALSE;
		bAWrappingCone123OnAuto:=FALSE;
		bAConeMissErrorAtWrpConvTemp2_24:=FALSE;
		TON_4_24(IN:=FALSE);
		TON_12_24(in:=FALSE);
		bWrapConvStopped2:=FALSE;
		bAConeMissErrorAtWrpConvTemp1_24:=FALSE;
 		TON_3(IN:=FALSE);
		TON_13_24(in:=FALSE);
		step1:=step1+2; END_IF

	9:	 IF bFilmErrClear THEN bSheetNotFeeded:='Continue Machine Operation';  bAFlimNotLoaded:=FALSE;bAConvRunning1:=FALSE;  step1:=step1+1;END_IF

	10:	 IF NOT bAPauseSeq  THEN  bAWrapConeCyl123:=FALSE;
		bA3ConeWrappOver_24:=TRUE;
		step1:=step1+1; END_IF

	11:	bFilmErrClear:=FALSE; TON_4_24(IN:=FALSE);
		TON_12_24(in:=FALSE);
		bWrapConvStopped2:=FALSE; step1:=step1+1;

	12:	 IF  bIWrappingChannelPiston1_Home   AND bIWrappingChannelPiston2_Home AND bIWrappingChannelPiston3_Home   THEN
		bASet1Comp:=TRUE;
		bAWrappingCone123FwdCom:=FALSE;
		bA3Pushed:=TRUE;
		bCount_ConvLockBit:=FALSE; SealingOver1:=FALSE;
		bAFilm1Loaded:=FALSE;
		bAFilm2Loaded:=FALSE;
		bAFilm3Loaded:=FALSE;
		bASet4Comp:=FALSE;
		WrapConvStartDly(in:=FALSE);
		bAConvRunning1:=FALSE;
		bWrapConvStopped2:=FALSE;
		TON_3(IN:=FALSE);
		TON_13_24(in:=FALSE);
		TON_4_24(IN:=FALSE);
		TON_12_24(in:=FALSE);
		bAConeMissErrorAtWrpConvTemp1_24:=FALSE;
		bAConeMissErrorAtWrpConvTemp2_24:=FALSE;
		bAWrapConeCyl123:=FALSE;
		step1:=0;
		END_IF   sMessage_Wrapping:='Check Wrapping Piston Home 1 & 2 & 3 Reed Switch';
END_CASE

IF bAFlimNotLoaded AND bErrorReset AND b2_4SetHmiSelected AND bAutoModeOn THEN step1:=10; bAFlimNotLoaded:=FALSE;HmiFilmLoadErr:=''; END_IF



                                                                (*===============Wrapping piston 3  ( 4th cone)  on/off logic  for 2*4 model====================*)


CASE step2 OF

	0:	TON_7(IN:= FALSE);
		step2:=step2+1;

	1:	 step2:=step2+1;

	2:	IF bAutoModeOn AND  bAWrapConeCyl3  AND SealingOver1  AND NOT bAFlimNotLoaded AND NOT bACheckWrappConvError3 AND b2_4SetHmiSelected
		  AND bIWrappingChannelPiston3_Home AND b2_4SetHmiSelected AND NOT bAResetEnabled  AND NOT bAConeMissErrorAtWrpConvTemp3_24
		AND SealingSafety THEN
		TON_7(IN:= TRUE, PT:=t#1s , Q=> , ET=> );
		 sMessage_Wrapping:='Check Wrapping Piston Home  3 Reed Switch';

		IF TON_7.Q THEN SealingOver1:=FALSE;	bASensorMonitorBit1:=FALSE;  step2:=step2+1; END_IF
		END_IF

	3:	step2:=step2+1;


	4:	IF NOT bQASealingConveyorMotor AND NOT bACheckWrappConvError3  AND NOT bQSealBitAlert (* AND NOT bQSealBitAlert_24*) AND NOT bAPauseSeq
		AND bIWrappingCone3   AND NOT bAConeMissErrorAtWrpConvTemp2_24   AND NOT bAConeMissErrorAtWrpConvTemp3_24
		 AND NOT bAConeMissErrorAtWrpConvTemp4_24  AND NOT bAConeMissErrorAtWrpConvTemp5_24    AND NOT SealConeMissAlet_24
		AND SealingSafety  THEN
		bAWrappingCone3OnAuto:=TRUE;
		bWrapConvStopped1_24exp:=FALSE;
		step2:=step2+1;
		END_IF

	5:	 step2:=step2+1;


	6:	IF bAWrappingCone3OnAuto AND bIWrappingChannelPiston3_End AND NOT bAWrap_PistRsError AND bAFilmLoadedCom
		 AND NOT bAConeMissErrorAtWrpConvTemp3_24 AND b2_4SetHmiSelected AND NOT bQSealBitAlert (*AND NOT bQSealBitAlert_24 *)  AND NOT SealConeMissAlet_24 THEN
		TON_7(IN:= FALSE);
		bAWrappingCone3FwdCom:=TRUE;
		bASensorMonitorBit1:=FALSE;
		bWrapConvStopped4_24exp:=FALSE;
		 TON_5_24(IN:=FALSE);
		TON_11_24(in:=FALSE);
		step2:=step2+1;
		ELSIF  bAWrappingCone3OnAuto AND bIWrappingChannelPiston3_End AND NOT bAWrap_PistRsError AND NOT bAFilmLoadedCom
		AND NOT bAPauseSeq  THEN
		bAFlimNotLoaded1:=TRUE;
		bAWrappingCone3OnAuto:=FALSE;
		bAWrapConeCyl3:=FALSE;
		bAPolythinSheetError:=TRUE;
		bAConeMissErrorAtWrpConvTemp3_24:=FALSE;
		bWrapConvStopped4_24exp:=FALSE;
 		TON_5_24(IN:=FALSE);
		TON_11_24(in:=FALSE);
		bSheetNotFeeded:='Sheet NOT Feeded'; step2:=step2+3; END_IF

	7:	step2:=step2+1;

	8: 	IF bAWrappingCone3FwdCom AND NOT bAPauseSeq  THEN
		bAWrappingCone3OnAuto:=FALSE;
		bAFilmLoadedCom:=FALSE;
		bASet1Comp:=FALSE; SealingOver1:=FALSE;
		bAConeMissErrorAtWrpConvTemp3_24:=FALSE;
		bWrapConvStopped4_24exp:=FALSE;
		 TON_5_24(IN:=FALSE);
		TON_11_24(in:=FALSE);
		step2:=step2+2;
		END_IF

	9:	 IF bFilmErrClear THEN bSheetNotFeeded:='Continue Machine Operation'; bAFlimNotLoaded1:=FALSE; bASensorMonitorBit1:=FALSE;  step2:=step2+1;END_IF


	10:	 IF NOT bAPauseSeq  THEN bAWrapConeCyl3:=FALSE;
		bA4thWrappOver:=TRUE;
		step2:=step2+1; END_IF

	11:	bFilmErrClear:=FALSE;bWrapConvStopped4_24exp:=FALSE;
		 TON_5_24(IN:=FALSE);
		TON_11_24(in:=FALSE);step2:=step2+1;

	12:	 IF  bIWrappingChannelPiston3_Home   THEN
		bASet2Comp:=TRUE;
		bAWrappingCone3FwdCom:=FALSE;
		b4thConePushed:=TRUE;
		bAFilm1Loaded_24_4Cone:=FALSE;
		bASensorMonitorBit1:=FALSE;
		bWrapConvStopped4_24exp:=FALSE;
 		TON_5_24(IN:=FALSE);
		TON_11_24(in:=FALSE);
		step2:=0;
		END_IF   sMessage_Wrapping:='Check Wrapping Piston Home  3 Reed Switch';
END_CASE


IF bAFlimNotLoaded1 AND b2_4SetHmiSelected AND bErrorReset AND bAutoModeOn THEN step2:=10; bAFlimNotLoaded1:=FALSE;HmiFilmLoadErr:=''; END_IF



                                                                            (*===============Wrapping piston 23 (Cone5,6 )on/off logic  for 2*4 model ====================*)
CASE step3 OF

	0:	TON_8(IN:= FALSE);
		step3:=step3+1;

	1:	 step3:=step3+1;

	2:	IF bAutoModeOn AND  bAWrapConeCyl23_24_1  AND SealingOver1 AND NOT bACheckWrappConvError4 AND NOT bAFlimNotLoaded1 AND b2_4SetHmiSelected
		 AND bIWrappingChannelPiston3_Home AND bIWrappingChannelPiston2_Home AND  b2_4SetHmiSelected  AND NOT bAResetEnabled AND SealingSafety
		AND NOT bAConeMissErrorAtWrpConvTemp4_24 THEN
		TON_8(IN:= TRUE, PT:=t#1s , Q=> , ET=> );
		 sMessage_Wrapping:='Check Wrapping Piston Home  2 & 3 Reed Switch';

		IF TON_8.Q THEN SealingOver1:=FALSE; bASensorMonitorBit2:=FALSE;  step3:=step3+1; END_IF
		END_IF

	3:	 step3:=step3+1;


	4:	IF NOT bQASealingConveyorMotor AND NOT bQSealBitAlert (*AND NOT bQSealBitAlert_24  *)AND bWCSStart2_24  AND NOT bAPauseSeq AND b2_4SetHmiSelected
		AND NOT bACheckWrappConvError4  AND  bIWrappingCone2 AND  bIWrappingCone3 AND NOT bAConeMissErrorAtWrpConvTemp4_24 AND NOT SealConeMissAlet_24
		AND SealingSafety THEN
		bAWrappingCone23OnAuto:=TRUE;
		step3:=step3+1;
		END_IF

	5:	 step3:=step3+1;

